REGION Network 41: FIT-503 LOW
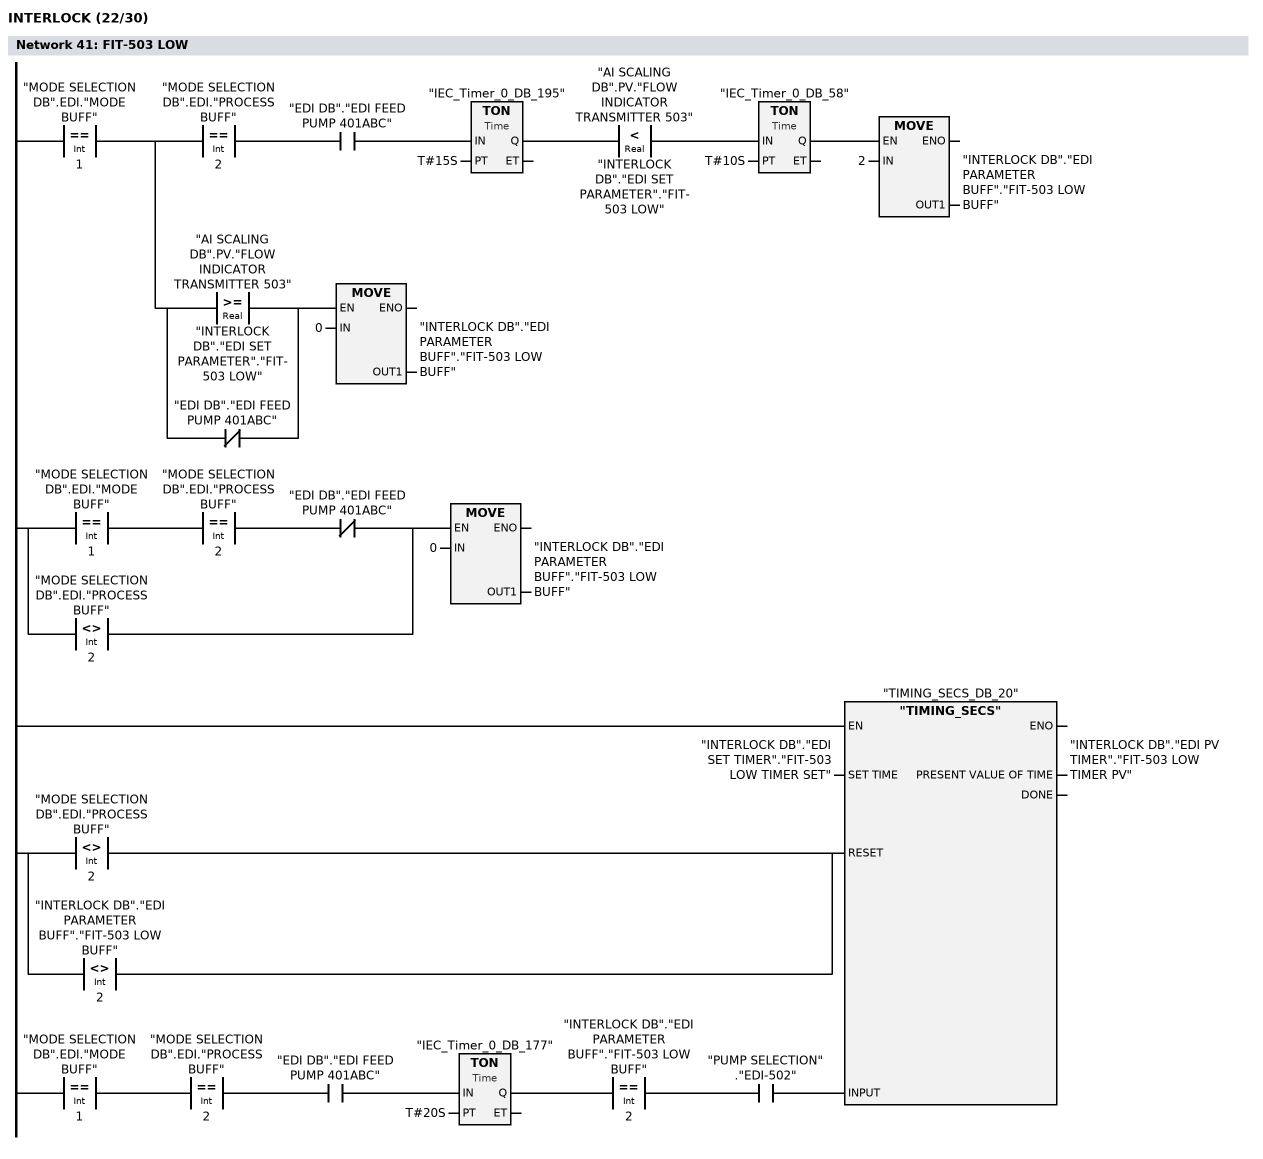
   RUNG wire#powerrail
      { S7_Templates := "SrcType := Int" } EQ_Contact(in1 := "MODE SELECTION DB".EDI."MODE BUFF", in2 := 1)
      wire#w1
      { S7_Templates := "SrcType := Int" } EQ_Contact(in1 := "MODE SELECTION DB".EDI."PROCESS BUFF", in2 := 2)
      Contact( "EDI DB"."EDI FEED PUMP 401ABC" )
      { S7_Templates := "time_type := Time" } "IEC_Timer_0_DB_195".TON(pt := T#15S, et =>)
      { S7_Templates := "SrcType := Real" } LT_Contact(in1 := "AI SCALING DB".PV."FLOW INDICATOR TRANSMITTER 503", in2 := "INTERLOCK DB"."EDI SET PARAMETER"."FIT-503 LOW")
      { S7_Templates := "time_type := Time" } "IEC_Timer_0_DB_58".TON(pt := T#10S, et =>)
      Move(in := 2, out1 => "INTERLOCK DB"."EDI PARAMETER BUFF"."FIT-503 LOW BUFF")
   END_RUNG
   RUNG wire#w1
      { S7_Templates := "SrcType := Real" } GE_Contact(in1 := "AI SCALING DB".PV."FLOW INDICATOR TRANSMITTER 503", in2 := "INTERLOCK DB"."EDI SET PARAMETER"."FIT-503 LOW")
      wire#w2
      Move(in := 0, out1 => "INTERLOCK DB"."EDI PARAMETER BUFF"."FIT-503 LOW BUFF")
   END_RUNG
   RUNG wire#w1
      I_Contact( "EDI DB"."EDI FEED PUMP 401ABC" )
   END_RUNG wire#w2
   RUNG wire#powerrail
      { S7_Templates := "SrcType := Int" } EQ_Contact(in1 := "MODE SELECTION DB".EDI."MODE BUFF", in2 := 1)
      { S7_Templates := "SrcType := Int" } EQ_Contact(in1 := "MODE SELECTION DB".EDI."PROCESS BUFF", in2 := 2)
      I_Contact( "EDI DB"."EDI FEED PUMP 401ABC" )
      wire#w3
      Move(in := 0, out1 => "INTERLOCK DB"."EDI PARAMETER BUFF"."FIT-503 LOW BUFF")
   END_RUNG
   RUNG wire#powerrail
      { S7_Templates := "SrcType := Int" } NE_Contact(in1 := "MODE SELECTION DB".EDI."PROCESS BUFF", in2 := 2)
   END_RUNG wire#w3
   RUNG wire#powerrail
      "TIMING_SECS_DB_20"(RESET := wire#w4, INPUT := wire#w5, "SET TIME" := "INTERLOCK DB"."EDI SET TIMER"."FIT-503 LOW TIMER SET", "PRESENT VALUE OF TIME" => "INTERLOCK DB"."EDI PV TIMER"."FIT-503 LOW TIMER PV", DONE =>)
   END_RUNG
   RUNG wire#powerrail
      { S7_Templates := "SrcType := Int" } NE_Contact(in1 := "MODE SELECTION DB".EDI."PROCESS BUFF", in2 := 2)
   END_RUNG wire#w4
   RUNG wire#powerrail
      { S7_Templates := "SrcType := Int" } NE_Contact(in1 := "INTERLOCK DB"."EDI PARAMETER BUFF"."FIT-503 LOW BUFF", in2 := 2)
   END_RUNG wire#w4
   RUNG wire#powerrail
      { S7_Templates := "SrcType := Int" } EQ_Contact(in1 := "MODE SELECTION DB".EDI."MODE BUFF", in2 := 1)
      { S7_Templates := "SrcType := Int" } EQ_Contact(in1 := "MODE SELECTION DB".EDI."PROCESS BUFF", in2 := 2)
      Contact( "EDI DB"."EDI FEED PUMP 401ABC" )
      { S7_Templates := "time_type := Time" } "IEC_Timer_0_DB_177".TON(pt := T#20S, et =>)
      { S7_Templates := "SrcType := Int" } EQ_Contact(in1 := "INTERLOCK DB"."EDI PARAMETER BUFF"."FIT-503 LOW BUFF", in2 := 2)
      Contact( "PUMP SELECTION"."EDI-502" )
   END_RUNG wire#w5
   // the same network as SCL:
   #_w1 := "MODE SELECTION DB".EDI."MODE BUFF" = 1;
   "IEC_Timer_0_DB_195".TON(IN := #_w1 AND ("MODE SELECTION DB".EDI."PROCESS BUFF" = 2) AND "EDI DB"."EDI FEED PUMP 401ABC",
                           PT := T#15S);
   "IEC_Timer_0_DB_58".TON(IN := "IEC_Timer_0_DB_195".Q AND ("AI SCALING DB".PV."FLOW INDICATOR TRANSMITTER 503" < "INTERLOCK DB"."EDI SET PARAMETER"."FIT-503 LOW"),
                           PT := T#10S);
   IF "IEC_Timer_0_DB_58".Q THEN "INTERLOCK DB"."EDI PARAMETER BUFF"."FIT-503 LOW BUFF" := 2; END_IF;
   IF #_w1 AND (("AI SCALING DB".PV."FLOW INDICATOR TRANSMITTER 503" >= "INTERLOCK DB"."EDI SET PARAMETER"."FIT-503 LOW") OR NOT "EDI DB"."EDI FEED PUMP 401ABC") THEN
       "INTERLOCK DB"."EDI PARAMETER BUFF"."FIT-503 LOW BUFF" := 0;
   END_IF;
   IF (("MODE SELECTION DB".EDI."MODE BUFF" = 1) AND ("MODE SELECTION DB".EDI."PROCESS BUFF" = 2) AND NOT "EDI DB"."EDI FEED PUMP 401ABC") OR ("MODE SELECTION DB".EDI."PROCESS BUFF" <> 2) THEN
       "INTERLOCK DB"."EDI PARAMETER BUFF"."FIT-503 LOW BUFF" := 0;
   END_IF;
   "IEC_Timer_0_DB_177".TON(IN := ("MODE SELECTION DB".EDI."MODE BUFF" = 1) AND ("MODE SELECTION DB".EDI."PROCESS BUFF" = 2) AND "EDI DB"."EDI FEED PUMP 401ABC",
                           PT := T#20S);
   "TIMING_SECS_DB_20"("SET TIME" := "INTERLOCK DB"."EDI SET TIMER"."FIT-503 LOW TIMER SET",   // "TIMING_SECS"
                       RESET := ("MODE SELECTION DB".EDI."PROCESS BUFF" <> 2) OR ("INTERLOCK DB"."EDI PARAMETER BUFF"."FIT-503 LOW BUFF" <> 2),
                       INPUT := "IEC_Timer_0_DB_177".Q AND ("INTERLOCK DB"."EDI PARAMETER BUFF"."FIT-503 LOW BUFF" = 2) AND "PUMP SELECTION"."EDI-502",
                       "PRESENT VALUE OF TIME" => "INTERLOCK DB"."EDI PV TIMER"."FIT-503 LOW TIMER PV");
END_REGION

REGION Network 42: FIT-504 LOW
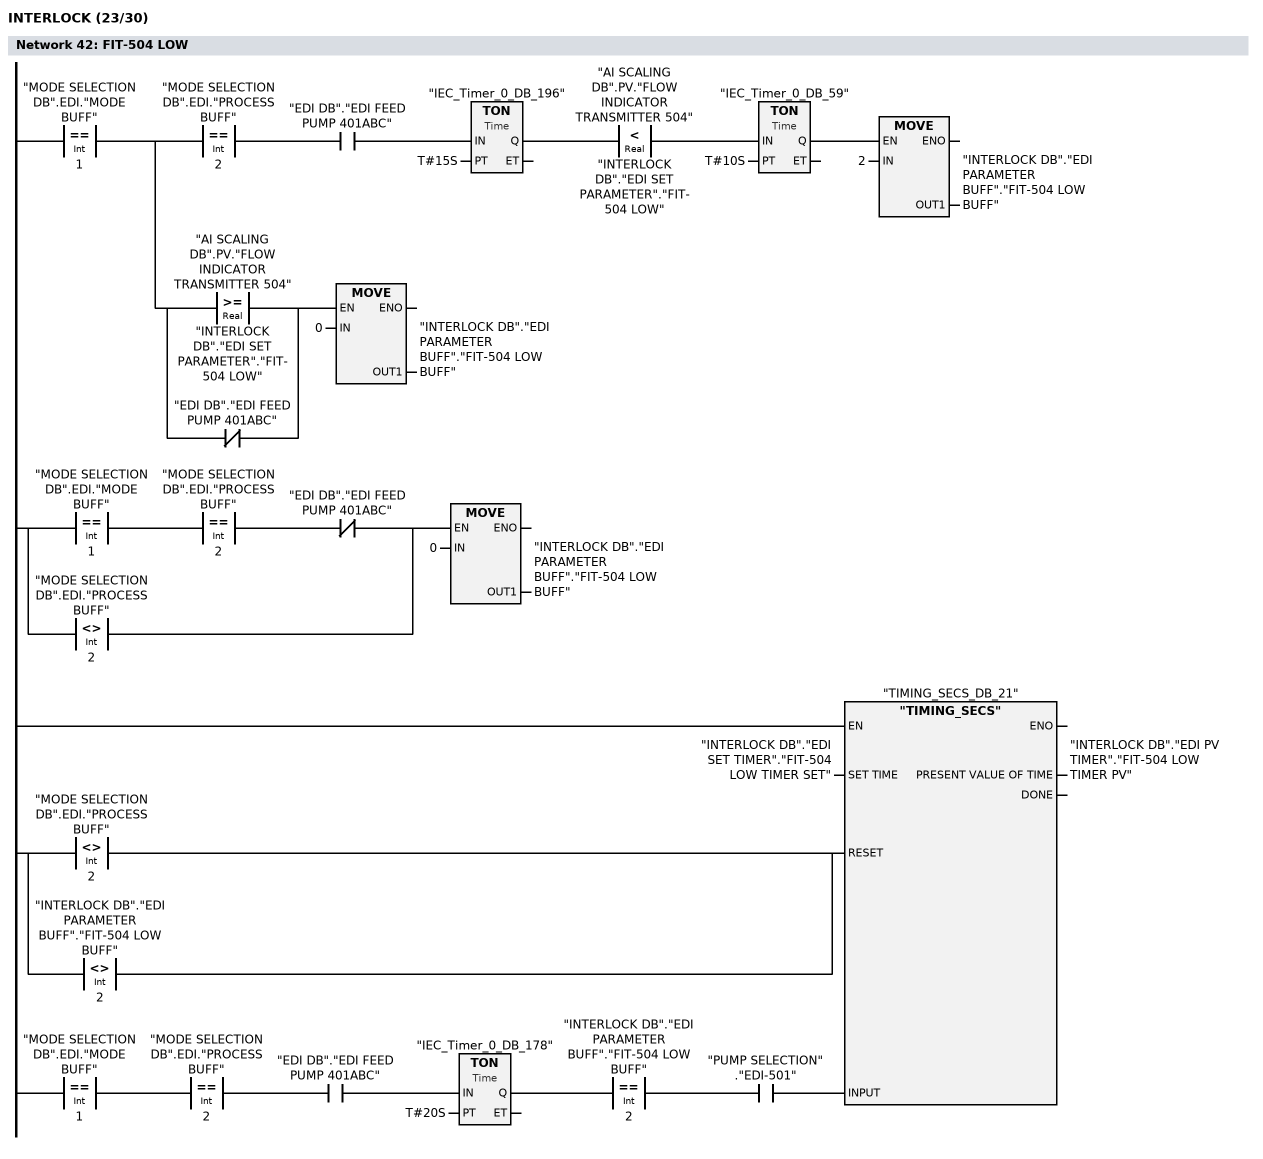
   RUNG wire#powerrail
      { S7_Templates := "SrcType := Int" } EQ_Contact(in1 := "MODE SELECTION DB".EDI."MODE BUFF", in2 := 1)
      wire#w1
      { S7_Templates := "SrcType := Int" } EQ_Contact(in1 := "MODE SELECTION DB".EDI."PROCESS BUFF", in2 := 2)
      Contact( "EDI DB"."EDI FEED PUMP 401ABC" )
      { S7_Templates := "time_type := Time" } "IEC_Timer_0_DB_196".TON(pt := T#15S, et =>)
      { S7_Templates := "SrcType := Real" } LT_Contact(in1 := "AI SCALING DB".PV."FLOW INDICATOR TRANSMITTER 504", in2 := "INTERLOCK DB"."EDI SET PARAMETER"."FIT-504 LOW")
      { S7_Templates := "time_type := Time" } "IEC_Timer_0_DB_59".TON(pt := T#10S, et =>)
      Move(in := 2, out1 => "INTERLOCK DB"."EDI PARAMETER BUFF"."FIT-504 LOW BUFF")
   END_RUNG
   RUNG wire#w1
      { S7_Templates := "SrcType := Real" } GE_Contact(in1 := "AI SCALING DB".PV."FLOW INDICATOR TRANSMITTER 504", in2 := "INTERLOCK DB"."EDI SET PARAMETER"."FIT-504 LOW")
      wire#w2
      Move(in := 0, out1 => "INTERLOCK DB"."EDI PARAMETER BUFF"."FIT-504 LOW BUFF")
   END_RUNG
   RUNG wire#w1
      I_Contact( "EDI DB"."EDI FEED PUMP 401ABC" )
   END_RUNG wire#w2
   RUNG wire#powerrail
      { S7_Templates := "SrcType := Int" } EQ_Contact(in1 := "MODE SELECTION DB".EDI."MODE BUFF", in2 := 1)
      { S7_Templates := "SrcType := Int" } EQ_Contact(in1 := "MODE SELECTION DB".EDI."PROCESS BUFF", in2 := 2)
      I_Contact( "EDI DB"."EDI FEED PUMP 401ABC" )
      wire#w3
      Move(in := 0, out1 => "INTERLOCK DB"."EDI PARAMETER BUFF"."FIT-504 LOW BUFF")
   END_RUNG
   RUNG wire#powerrail
      { S7_Templates := "SrcType := Int" } NE_Contact(in1 := "MODE SELECTION DB".EDI."PROCESS BUFF", in2 := 2)
   END_RUNG wire#w3
   RUNG wire#powerrail
      "TIMING_SECS_DB_21"(RESET := wire#w4, INPUT := wire#w5, "SET TIME" := "INTERLOCK DB"."EDI SET TIMER"."FIT-504 LOW TIMER SET", "PRESENT VALUE OF TIME" => "INTERLOCK DB"."EDI PV TIMER"."FIT-504 LOW TIMER PV", DONE =>)
   END_RUNG
   RUNG wire#powerrail
      { S7_Templates := "SrcType := Int" } NE_Contact(in1 := "MODE SELECTION DB".EDI."PROCESS BUFF", in2 := 2)
   END_RUNG wire#w4
   RUNG wire#powerrail
      { S7_Templates := "SrcType := Int" } NE_Contact(in1 := "INTERLOCK DB"."EDI PARAMETER BUFF"."FIT-504 LOW BUFF", in2 := 2)
   END_RUNG wire#w4
   RUNG wire#powerrail
      { S7_Templates := "SrcType := Int" } EQ_Contact(in1 := "MODE SELECTION DB".EDI."MODE BUFF", in2 := 1)
      { S7_Templates := "SrcType := Int" } EQ_Contact(in1 := "MODE SELECTION DB".EDI."PROCESS BUFF", in2 := 2)
      Contact( "EDI DB"."EDI FEED PUMP 401ABC" )
      { S7_Templates := "time_type := Time" } "IEC_Timer_0_DB_178".TON(pt := T#20S, et =>)
      { S7_Templates := "SrcType := Int" } EQ_Contact(in1 := "INTERLOCK DB"."EDI PARAMETER BUFF"."FIT-504 LOW BUFF", in2 := 2)
      Contact( "PUMP SELECTION"."EDI-501" )
   END_RUNG wire#w5
   // the same network as SCL:
   #_w1 := "MODE SELECTION DB".EDI."MODE BUFF" = 1;
   "IEC_Timer_0_DB_196".TON(IN := #_w1 AND ("MODE SELECTION DB".EDI."PROCESS BUFF" = 2) AND "EDI DB"."EDI FEED PUMP 401ABC",
                           PT := T#15S);
   "IEC_Timer_0_DB_59".TON(IN := "IEC_Timer_0_DB_196".Q AND ("AI SCALING DB".PV."FLOW INDICATOR TRANSMITTER 504" < "INTERLOCK DB"."EDI SET PARAMETER"."FIT-504 LOW"),
                           PT := T#10S);
   IF "IEC_Timer_0_DB_59".Q THEN "INTERLOCK DB"."EDI PARAMETER BUFF"."FIT-504 LOW BUFF" := 2; END_IF;
   IF #_w1 AND (("AI SCALING DB".PV."FLOW INDICATOR TRANSMITTER 504" >= "INTERLOCK DB"."EDI SET PARAMETER"."FIT-504 LOW") OR NOT "EDI DB"."EDI FEED PUMP 401ABC") THEN
       "INTERLOCK DB"."EDI PARAMETER BUFF"."FIT-504 LOW BUFF" := 0;
   END_IF;
   IF (("MODE SELECTION DB".EDI."MODE BUFF" = 1) AND ("MODE SELECTION DB".EDI."PROCESS BUFF" = 2) AND NOT "EDI DB"."EDI FEED PUMP 401ABC") OR ("MODE SELECTION DB".EDI."PROCESS BUFF" <> 2) THEN
       "INTERLOCK DB"."EDI PARAMETER BUFF"."FIT-504 LOW BUFF" := 0;
   END_IF;
   "IEC_Timer_0_DB_178".TON(IN := ("MODE SELECTION DB".EDI."MODE BUFF" = 1) AND ("MODE SELECTION DB".EDI."PROCESS BUFF" = 2) AND "EDI DB"."EDI FEED PUMP 401ABC",
                           PT := T#20S);
   "TIMING_SECS_DB_21"("SET TIME" := "INTERLOCK DB"."EDI SET TIMER"."FIT-504 LOW TIMER SET",   // "TIMING_SECS"
                       RESET := ("MODE SELECTION DB".EDI."PROCESS BUFF" <> 2) OR ("INTERLOCK DB"."EDI PARAMETER BUFF"."FIT-504 LOW BUFF" <> 2),
                       INPUT := "IEC_Timer_0_DB_178".Q AND ("INTERLOCK DB"."EDI PARAMETER BUFF"."FIT-504 LOW BUFF" = 2) AND "PUMP SELECTION"."EDI-501",
                       "PRESENT VALUE OF TIME" => "INTERLOCK DB"."EDI PV TIMER"."FIT-504 LOW TIMER PV");
END_REGION

REGION Network 43: FIT-505 LOW / HIGH
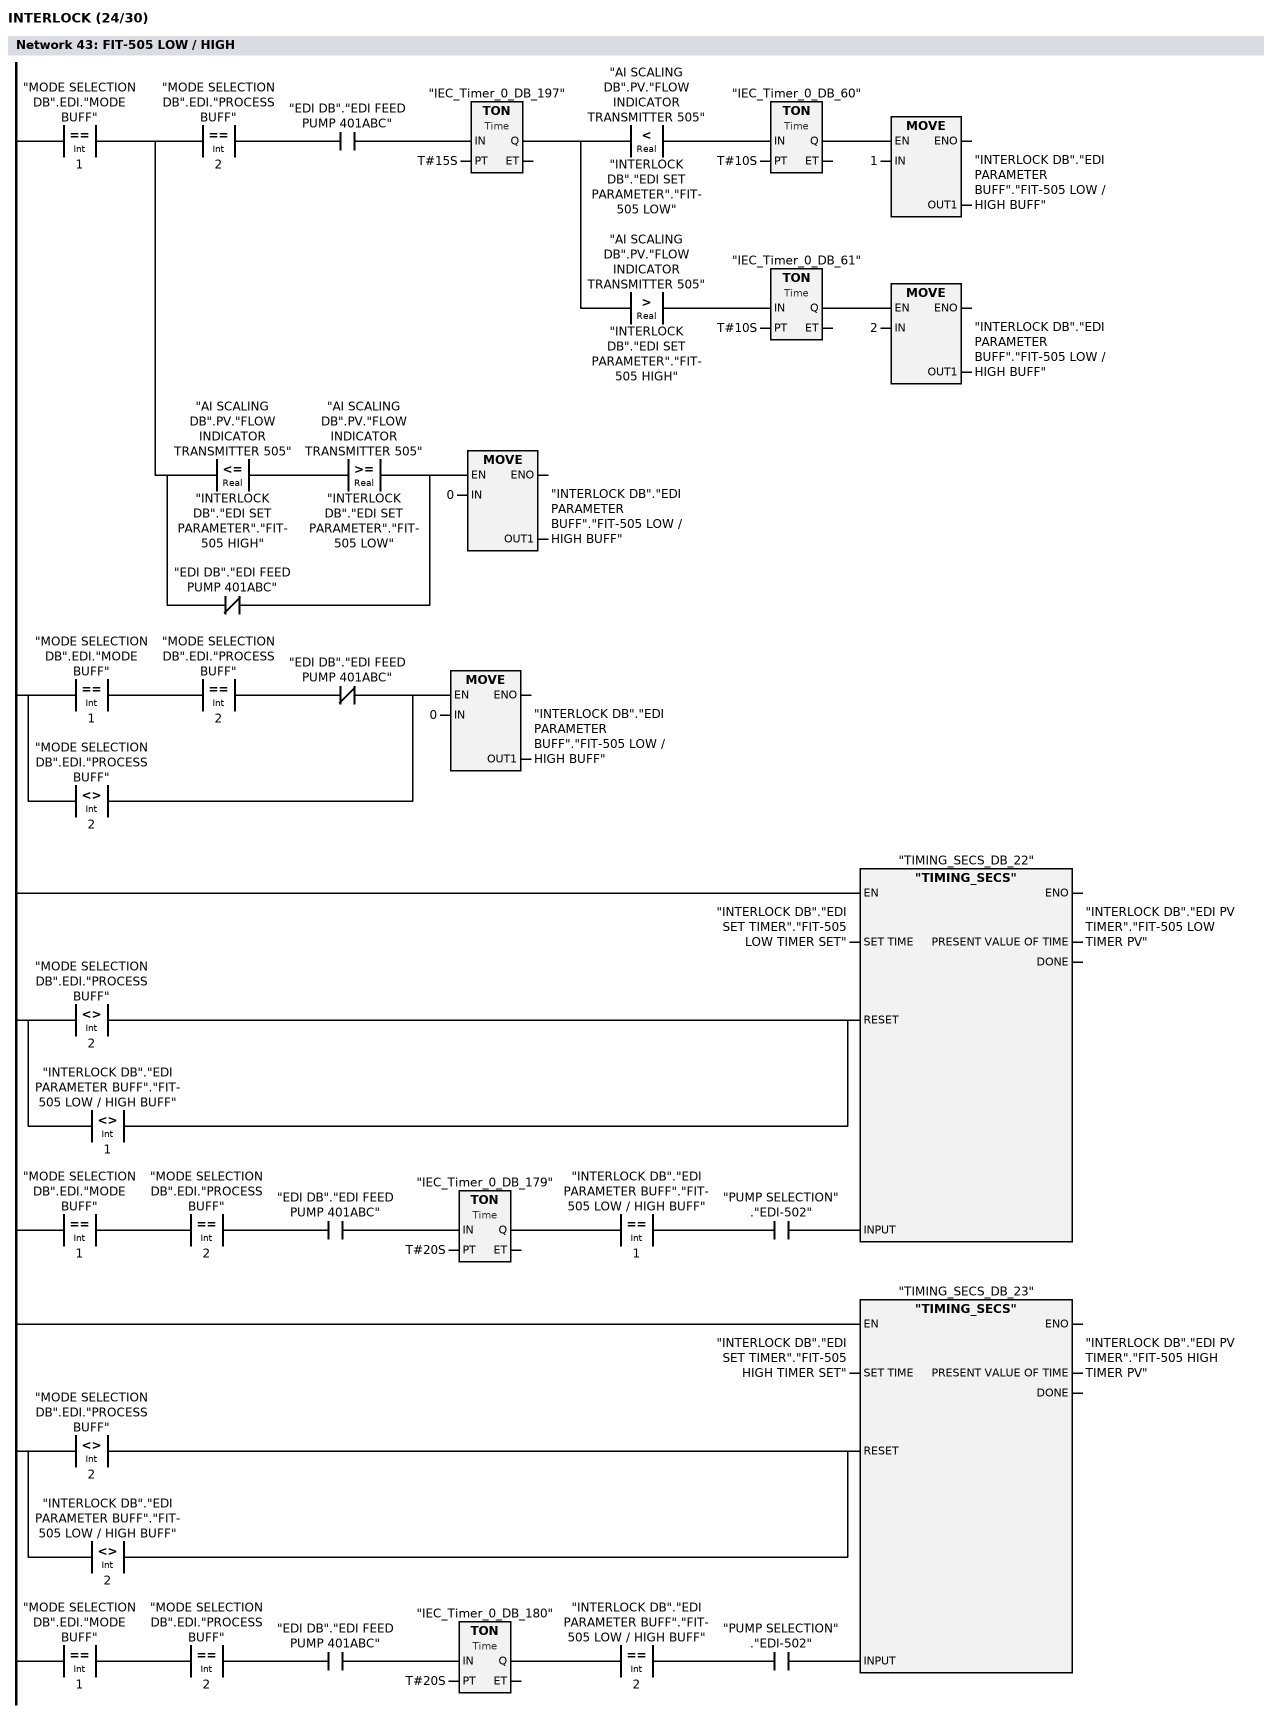
   RUNG wire#powerrail
      { S7_Templates := "SrcType := Int" } EQ_Contact(in1 := "MODE SELECTION DB".EDI."MODE BUFF", in2 := 1)
      wire#w1
      { S7_Templates := "SrcType := Int" } EQ_Contact(in1 := "MODE SELECTION DB".EDI."PROCESS BUFF", in2 := 2)
      Contact( "EDI DB"."EDI FEED PUMP 401ABC" )
      { S7_Templates := "time_type := Time" } "IEC_Timer_0_DB_197".TON(pt := T#15S, et =>)
      wire#w2
      { S7_Templates := "SrcType := Real" } LT_Contact(in1 := "AI SCALING DB".PV."FLOW INDICATOR TRANSMITTER 505", in2 := "INTERLOCK DB"."EDI SET PARAMETER"."FIT-505 LOW")
      { S7_Templates := "time_type := Time" } "IEC_Timer_0_DB_60".TON(pt := T#10S, et =>)
      Move(in := 1, out1 => "INTERLOCK DB"."EDI PARAMETER BUFF"."FIT-505 LOW / HIGH BUFF")
   END_RUNG
   RUNG wire#w2
      { S7_Templates := "SrcType := Real" } GT_Contact(in1 := "AI SCALING DB".PV."FLOW INDICATOR TRANSMITTER 505", in2 := "INTERLOCK DB"."EDI SET PARAMETER"."FIT-505 HIGH")
      { S7_Templates := "time_type := Time" } "IEC_Timer_0_DB_61".TON(pt := T#10S, et =>)
      Move(in := 2, out1 => "INTERLOCK DB"."EDI PARAMETER BUFF"."FIT-505 LOW / HIGH BUFF")
   END_RUNG
   RUNG wire#w1
      { S7_Templates := "SrcType := Real" } LE_Contact(in1 := "AI SCALING DB".PV."FLOW INDICATOR TRANSMITTER 505", in2 := "INTERLOCK DB"."EDI SET PARAMETER"."FIT-505 HIGH")
      { S7_Templates := "SrcType := Real" } GE_Contact(in1 := "AI SCALING DB".PV."FLOW INDICATOR TRANSMITTER 505", in2 := "INTERLOCK DB"."EDI SET PARAMETER"."FIT-505 LOW")
      wire#w3
      Move(in := 0, out1 => "INTERLOCK DB"."EDI PARAMETER BUFF"."FIT-505 LOW / HIGH BUFF")
   END_RUNG
   RUNG wire#w1
      I_Contact( "EDI DB"."EDI FEED PUMP 401ABC" )
   END_RUNG wire#w3
   RUNG wire#powerrail
      { S7_Templates := "SrcType := Int" } EQ_Contact(in1 := "MODE SELECTION DB".EDI."MODE BUFF", in2 := 1)
      { S7_Templates := "SrcType := Int" } EQ_Contact(in1 := "MODE SELECTION DB".EDI."PROCESS BUFF", in2 := 2)
      I_Contact( "EDI DB"."EDI FEED PUMP 401ABC" )
      wire#w4
      Move(in := 0, out1 => "INTERLOCK DB"."EDI PARAMETER BUFF"."FIT-505 LOW / HIGH BUFF")
   END_RUNG
   RUNG wire#powerrail
      { S7_Templates := "SrcType := Int" } NE_Contact(in1 := "MODE SELECTION DB".EDI."PROCESS BUFF", in2 := 2)
   END_RUNG wire#w4
   RUNG wire#powerrail
      "TIMING_SECS_DB_22"(RESET := wire#w5, INPUT := wire#w6, "SET TIME" := "INTERLOCK DB"."EDI SET TIMER"."FIT-505 LOW TIMER SET", "PRESENT VALUE OF TIME" => "INTERLOCK DB"."EDI PV TIMER"."FIT-505 LOW TIMER PV", DONE =>)
   END_RUNG
   RUNG wire#powerrail
      { S7_Templates := "SrcType := Int" } NE_Contact(in1 := "MODE SELECTION DB".EDI."PROCESS BUFF", in2 := 2)
   END_RUNG wire#w5
   RUNG wire#powerrail
      { S7_Templates := "SrcType := Int" } NE_Contact(in1 := "INTERLOCK DB"."EDI PARAMETER BUFF"."FIT-505 LOW / HIGH BUFF", in2 := 1)
   END_RUNG wire#w5
   RUNG wire#powerrail
      { S7_Templates := "SrcType := Int" } EQ_Contact(in1 := "MODE SELECTION DB".EDI."MODE BUFF", in2 := 1)
      { S7_Templates := "SrcType := Int" } EQ_Contact(in1 := "MODE SELECTION DB".EDI."PROCESS BUFF", in2 := 2)
      Contact( "EDI DB"."EDI FEED PUMP 401ABC" )
      { S7_Templates := "time_type := Time" } "IEC_Timer_0_DB_179".TON(pt := T#20S, et =>)
      { S7_Templates := "SrcType := Int" } EQ_Contact(in1 := "INTERLOCK DB"."EDI PARAMETER BUFF"."FIT-505 LOW / HIGH BUFF", in2 := 1)
      Contact( "PUMP SELECTION"."EDI-502" )
   END_RUNG wire#w6
   RUNG wire#powerrail
      "TIMING_SECS_DB_23"(RESET := wire#w7, INPUT := wire#w8, "SET TIME" := "INTERLOCK DB"."EDI SET TIMER"."FIT-505 HIGH TIMER SET", "PRESENT VALUE OF TIME" => "INTERLOCK DB"."EDI PV TIMER"."FIT-505 HIGH TIMER PV", DONE =>)
   END_RUNG
   RUNG wire#powerrail
      { S7_Templates := "SrcType := Int" } NE_Contact(in1 := "MODE SELECTION DB".EDI."PROCESS BUFF", in2 := 2)
   END_RUNG wire#w7
   RUNG wire#powerrail
      { S7_Templates := "SrcType := Int" } NE_Contact(in1 := "INTERLOCK DB"."EDI PARAMETER BUFF"."FIT-505 LOW / HIGH BUFF", in2 := 2)
   END_RUNG wire#w7
   RUNG wire#powerrail
      { S7_Templates := "SrcType := Int" } EQ_Contact(in1 := "MODE SELECTION DB".EDI."MODE BUFF", in2 := 1)
      { S7_Templates := "SrcType := Int" } EQ_Contact(in1 := "MODE SELECTION DB".EDI."PROCESS BUFF", in2 := 2)
      Contact( "EDI DB"."EDI FEED PUMP 401ABC" )
      { S7_Templates := "time_type := Time" } "IEC_Timer_0_DB_180".TON(pt := T#20S, et =>)
      { S7_Templates := "SrcType := Int" } EQ_Contact(in1 := "INTERLOCK DB"."EDI PARAMETER BUFF"."FIT-505 LOW / HIGH BUFF", in2 := 2)
      Contact( "PUMP SELECTION"."EDI-502" )
   END_RUNG wire#w8
   // the same network as SCL:
   #_w1 := "MODE SELECTION DB".EDI."MODE BUFF" = 1;
   "IEC_Timer_0_DB_197".TON(IN := #_w1 AND ("MODE SELECTION DB".EDI."PROCESS BUFF" = 2) AND "EDI DB"."EDI FEED PUMP 401ABC",
                           PT := T#15S);
   "IEC_Timer_0_DB_60".TON(IN := "IEC_Timer_0_DB_197".Q AND ("AI SCALING DB".PV."FLOW INDICATOR TRANSMITTER 505" < "INTERLOCK DB"."EDI SET PARAMETER"."FIT-505 LOW"),
                           PT := T#10S);
   IF "IEC_Timer_0_DB_60".Q THEN "INTERLOCK DB"."EDI PARAMETER BUFF"."FIT-505 LOW / HIGH BUFF" := 1; END_IF;
   "IEC_Timer_0_DB_61".TON(IN := "IEC_Timer_0_DB_197".Q AND ("AI SCALING DB".PV."FLOW INDICATOR TRANSMITTER 505" > "INTERLOCK DB"."EDI SET PARAMETER"."FIT-505 HIGH"),
                           PT := T#10S);
   IF "IEC_Timer_0_DB_61".Q THEN "INTERLOCK DB"."EDI PARAMETER BUFF"."FIT-505 LOW / HIGH BUFF" := 2; END_IF;
   IF #_w1 AND ((("AI SCALING DB".PV."FLOW INDICATOR TRANSMITTER 505" <= "INTERLOCK DB"."EDI SET PARAMETER"."FIT-505 HIGH") AND ("AI SCALING DB".PV."FLOW INDICATOR TRANSMITTER 505" >= "INTERLOCK DB"."EDI SET PARAMETER"."FIT-505 LOW")) OR NOT "EDI DB"."EDI FEED PUMP 401ABC") THEN
       "INTERLOCK DB"."EDI PARAMETER BUFF"."FIT-505 LOW / HIGH BUFF" := 0;
   END_IF;
   IF (("MODE SELECTION DB".EDI."MODE BUFF" = 1) AND ("MODE SELECTION DB".EDI."PROCESS BUFF" = 2) AND NOT "EDI DB"."EDI FEED PUMP 401ABC") OR ("MODE SELECTION DB".EDI."PROCESS BUFF" <> 2) THEN
       "INTERLOCK DB"."EDI PARAMETER BUFF"."FIT-505 LOW / HIGH BUFF" := 0;
   END_IF;
   "IEC_Timer_0_DB_179".TON(IN := ("MODE SELECTION DB".EDI."MODE BUFF" = 1) AND ("MODE SELECTION DB".EDI."PROCESS BUFF" = 2) AND "EDI DB"."EDI FEED PUMP 401ABC",
                           PT := T#20S);
   "TIMING_SECS_DB_22"("SET TIME" := "INTERLOCK DB"."EDI SET TIMER"."FIT-505 LOW TIMER SET",   // "TIMING_SECS"
                       RESET := ("MODE SELECTION DB".EDI."PROCESS BUFF" <> 2) OR ("INTERLOCK DB"."EDI PARAMETER BUFF"."FIT-505 LOW / HIGH BUFF" <> 1),
                       INPUT := "IEC_Timer_0_DB_179".Q AND ("INTERLOCK DB"."EDI PARAMETER BUFF"."FIT-505 LOW / HIGH BUFF" = 1) AND "PUMP SELECTION"."EDI-502",
                       "PRESENT VALUE OF TIME" => "INTERLOCK DB"."EDI PV TIMER"."FIT-505 LOW TIMER PV");
   "IEC_Timer_0_DB_180".TON(IN := ("MODE SELECTION DB".EDI."MODE BUFF" = 1) AND ("MODE SELECTION DB".EDI."PROCESS BUFF" = 2) AND "EDI DB"."EDI FEED PUMP 401ABC",
                           PT := T#20S);
   "TIMING_SECS_DB_23"("SET TIME" := "INTERLOCK DB"."EDI SET TIMER"."FIT-505 HIGH TIMER SET",   // "TIMING_SECS"
                       RESET := ("MODE SELECTION DB".EDI."PROCESS BUFF" <> 2) OR ("INTERLOCK DB"."EDI PARAMETER BUFF"."FIT-505 LOW / HIGH BUFF" <> 2),
                       INPUT := "IEC_Timer_0_DB_180".Q AND ("INTERLOCK DB"."EDI PARAMETER BUFF"."FIT-505 LOW / HIGH BUFF" = 2) AND "PUMP SELECTION"."EDI-502",
                       "PRESENT VALUE OF TIME" => "INTERLOCK DB"."EDI PV TIMER"."FIT-505 HIGH TIMER PV");
END_REGION

REGION Network 44: FIT-506 LOW / HIGH
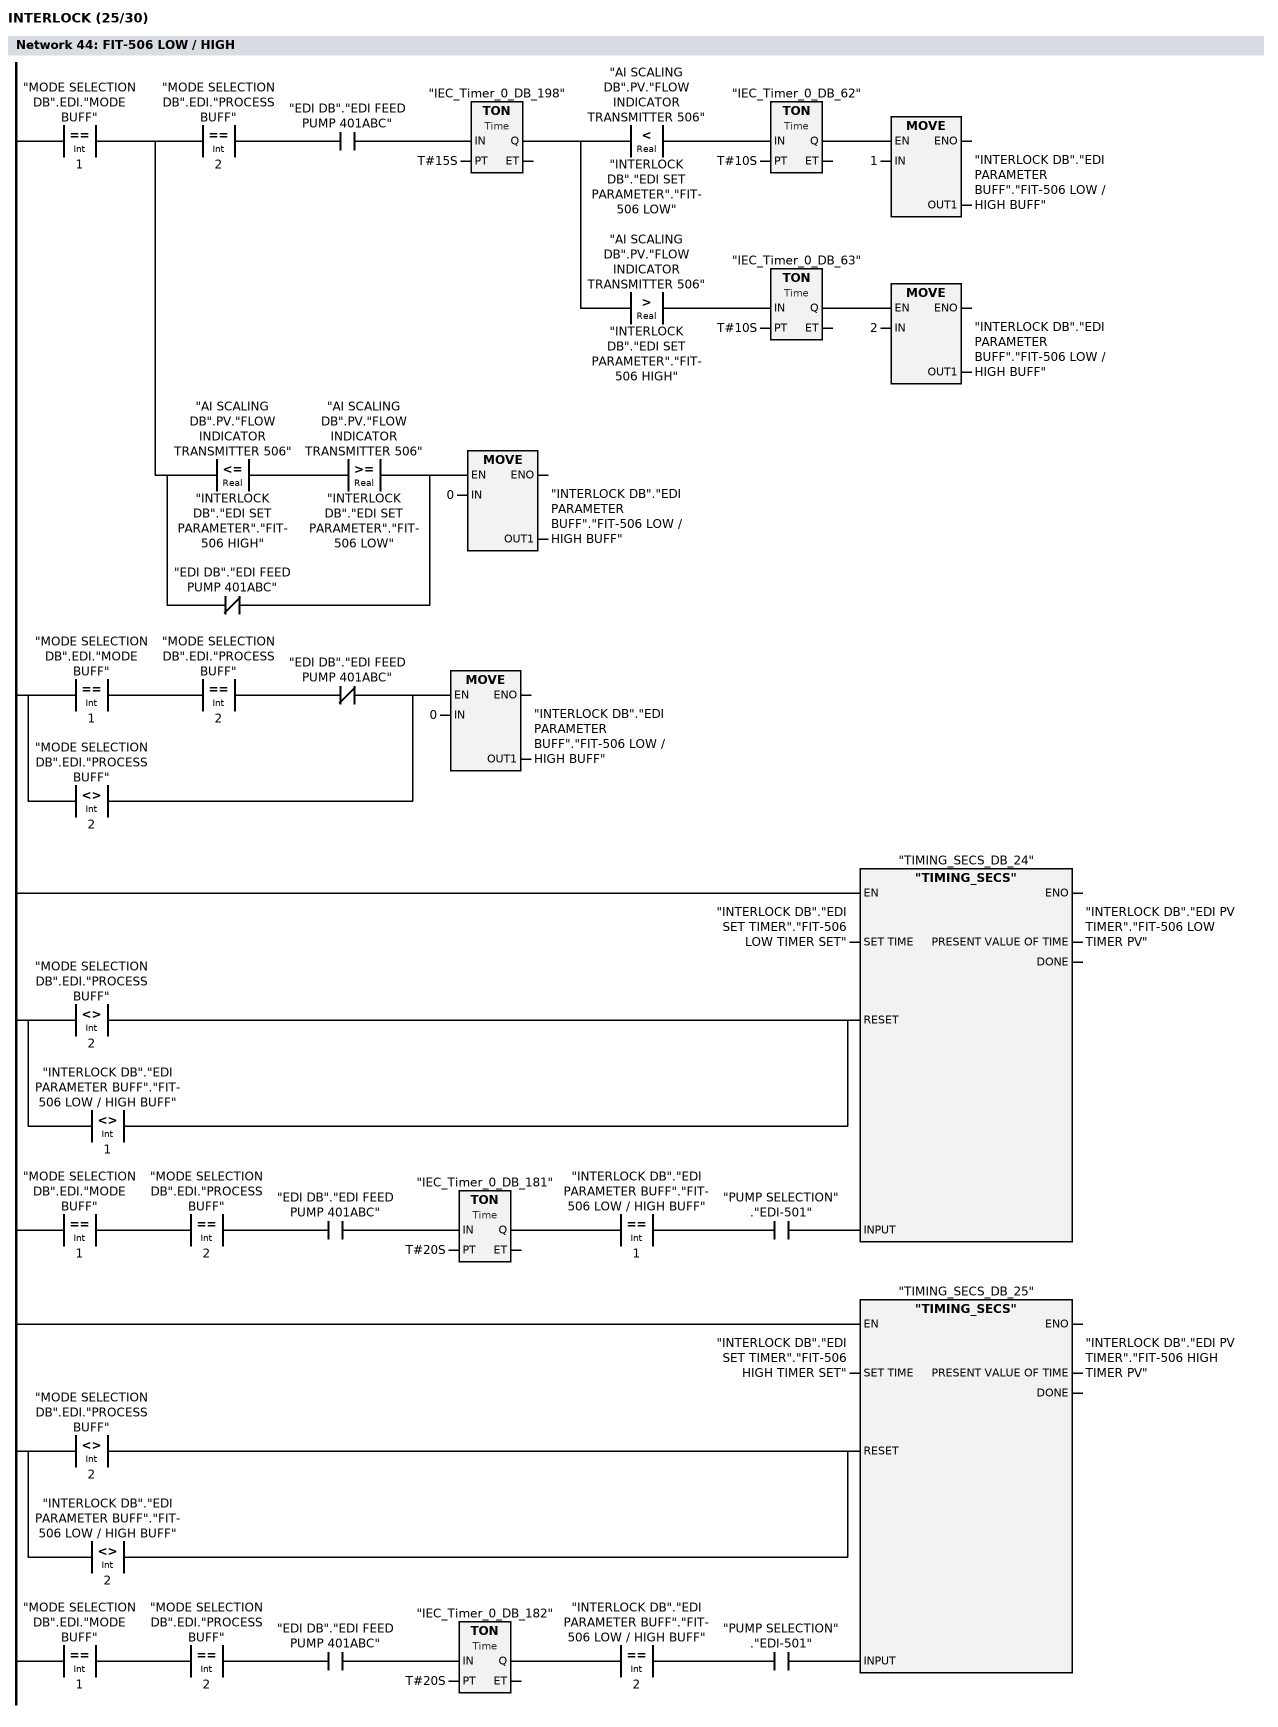
   RUNG wire#powerrail
      { S7_Templates := "SrcType := Int" } EQ_Contact(in1 := "MODE SELECTION DB".EDI."MODE BUFF", in2 := 1)
      wire#w1
      { S7_Templates := "SrcType := Int" } EQ_Contact(in1 := "MODE SELECTION DB".EDI."PROCESS BUFF", in2 := 2)
      Contact( "EDI DB"."EDI FEED PUMP 401ABC" )
      { S7_Templates := "time_type := Time" } "IEC_Timer_0_DB_198".TON(pt := T#15S, et =>)
      wire#w2
      { S7_Templates := "SrcType := Real" } LT_Contact(in1 := "AI SCALING DB".PV."FLOW INDICATOR TRANSMITTER 506", in2 := "INTERLOCK DB"."EDI SET PARAMETER"."FIT-506 LOW")
      { S7_Templates := "time_type := Time" } "IEC_Timer_0_DB_62".TON(pt := T#10S, et =>)
      Move(in := 1, out1 => "INTERLOCK DB"."EDI PARAMETER BUFF"."FIT-506 LOW / HIGH BUFF")
   END_RUNG
   RUNG wire#w2
      { S7_Templates := "SrcType := Real" } GT_Contact(in1 := "AI SCALING DB".PV."FLOW INDICATOR TRANSMITTER 506", in2 := "INTERLOCK DB"."EDI SET PARAMETER"."FIT-506 HIGH")
      { S7_Templates := "time_type := Time" } "IEC_Timer_0_DB_63".TON(pt := T#10S, et =>)
      Move(in := 2, out1 => "INTERLOCK DB"."EDI PARAMETER BUFF"."FIT-506 LOW / HIGH BUFF")
   END_RUNG
   RUNG wire#w1
      { S7_Templates := "SrcType := Real" } LE_Contact(in1 := "AI SCALING DB".PV."FLOW INDICATOR TRANSMITTER 506", in2 := "INTERLOCK DB"."EDI SET PARAMETER"."FIT-506 HIGH")
      { S7_Templates := "SrcType := Real" } GE_Contact(in1 := "AI SCALING DB".PV."FLOW INDICATOR TRANSMITTER 506", in2 := "INTERLOCK DB"."EDI SET PARAMETER"."FIT-506 LOW")
      wire#w3
      Move(in := 0, out1 => "INTERLOCK DB"."EDI PARAMETER BUFF"."FIT-506 LOW / HIGH BUFF")
   END_RUNG
   RUNG wire#w1
      I_Contact( "EDI DB"."EDI FEED PUMP 401ABC" )
   END_RUNG wire#w3
   RUNG wire#powerrail
      { S7_Templates := "SrcType := Int" } EQ_Contact(in1 := "MODE SELECTION DB".EDI."MODE BUFF", in2 := 1)
      { S7_Templates := "SrcType := Int" } EQ_Contact(in1 := "MODE SELECTION DB".EDI."PROCESS BUFF", in2 := 2)
      I_Contact( "EDI DB"."EDI FEED PUMP 401ABC" )
      wire#w4
      Move(in := 0, out1 => "INTERLOCK DB"."EDI PARAMETER BUFF"."FIT-506 LOW / HIGH BUFF")
   END_RUNG
   RUNG wire#powerrail
      { S7_Templates := "SrcType := Int" } NE_Contact(in1 := "MODE SELECTION DB".EDI."PROCESS BUFF", in2 := 2)
   END_RUNG wire#w4
   RUNG wire#powerrail
      "TIMING_SECS_DB_24"(RESET := wire#w5, INPUT := wire#w6, "SET TIME" := "INTERLOCK DB"."EDI SET TIMER"."FIT-506 LOW TIMER SET", "PRESENT VALUE OF TIME" => "INTERLOCK DB"."EDI PV TIMER"."FIT-506 LOW TIMER PV", DONE =>)
   END_RUNG
   RUNG wire#powerrail
      { S7_Templates := "SrcType := Int" } NE_Contact(in1 := "MODE SELECTION DB".EDI."PROCESS BUFF", in2 := 2)
   END_RUNG wire#w5
   RUNG wire#powerrail
      { S7_Templates := "SrcType := Int" } NE_Contact(in1 := "INTERLOCK DB"."EDI PARAMETER BUFF"."FIT-506 LOW / HIGH BUFF", in2 := 1)
   END_RUNG wire#w5
   RUNG wire#powerrail
      { S7_Templates := "SrcType := Int" } EQ_Contact(in1 := "MODE SELECTION DB".EDI."MODE BUFF", in2 := 1)
      { S7_Templates := "SrcType := Int" } EQ_Contact(in1 := "MODE SELECTION DB".EDI."PROCESS BUFF", in2 := 2)
      Contact( "EDI DB"."EDI FEED PUMP 401ABC" )
      { S7_Templates := "time_type := Time" } "IEC_Timer_0_DB_181".TON(pt := T#20S, et =>)
      { S7_Templates := "SrcType := Int" } EQ_Contact(in1 := "INTERLOCK DB"."EDI PARAMETER BUFF"."FIT-506 LOW / HIGH BUFF", in2 := 1)
      Contact( "PUMP SELECTION"."EDI-501" )
   END_RUNG wire#w6
   RUNG wire#powerrail
      "TIMING_SECS_DB_25"(RESET := wire#w7, INPUT := wire#w8, "SET TIME" := "INTERLOCK DB"."EDI SET TIMER"."FIT-506 HIGH TIMER SET", "PRESENT VALUE OF TIME" => "INTERLOCK DB"."EDI PV TIMER"."FIT-506 HIGH TIMER PV", DONE =>)
   END_RUNG
   RUNG wire#powerrail
      { S7_Templates := "SrcType := Int" } NE_Contact(in1 := "MODE SELECTION DB".EDI."PROCESS BUFF", in2 := 2)
   END_RUNG wire#w7
   RUNG wire#powerrail
      { S7_Templates := "SrcType := Int" } NE_Contact(in1 := "INTERLOCK DB"."EDI PARAMETER BUFF"."FIT-506 LOW / HIGH BUFF", in2 := 2)
   END_RUNG wire#w7
   RUNG wire#powerrail
      { S7_Templates := "SrcType := Int" } EQ_Contact(in1 := "MODE SELECTION DB".EDI."MODE BUFF", in2 := 1)
      { S7_Templates := "SrcType := Int" } EQ_Contact(in1 := "MODE SELECTION DB".EDI."PROCESS BUFF", in2 := 2)
      Contact( "EDI DB"."EDI FEED PUMP 401ABC" )
      { S7_Templates := "time_type := Time" } "IEC_Timer_0_DB_182".TON(pt := T#20S, et =>)
      { S7_Templates := "SrcType := Int" } EQ_Contact(in1 := "INTERLOCK DB"."EDI PARAMETER BUFF"."FIT-506 LOW / HIGH BUFF", in2 := 2)
      Contact( "PUMP SELECTION"."EDI-501" )
   END_RUNG wire#w8
   // the same network as SCL:
   #_w1 := "MODE SELECTION DB".EDI."MODE BUFF" = 1;
   "IEC_Timer_0_DB_198".TON(IN := #_w1 AND ("MODE SELECTION DB".EDI."PROCESS BUFF" = 2) AND "EDI DB"."EDI FEED PUMP 401ABC",
                           PT := T#15S);
   "IEC_Timer_0_DB_62".TON(IN := "IEC_Timer_0_DB_198".Q AND ("AI SCALING DB".PV."FLOW INDICATOR TRANSMITTER 506" < "INTERLOCK DB"."EDI SET PARAMETER"."FIT-506 LOW"),
                           PT := T#10S);
   IF "IEC_Timer_0_DB_62".Q THEN "INTERLOCK DB"."EDI PARAMETER BUFF"."FIT-506 LOW / HIGH BUFF" := 1; END_IF;
   "IEC_Timer_0_DB_63".TON(IN := "IEC_Timer_0_DB_198".Q AND ("AI SCALING DB".PV."FLOW INDICATOR TRANSMITTER 506" > "INTERLOCK DB"."EDI SET PARAMETER"."FIT-506 HIGH"),
                           PT := T#10S);
   IF "IEC_Timer_0_DB_63".Q THEN "INTERLOCK DB"."EDI PARAMETER BUFF"."FIT-506 LOW / HIGH BUFF" := 2; END_IF;
   IF #_w1 AND ((("AI SCALING DB".PV."FLOW INDICATOR TRANSMITTER 506" <= "INTERLOCK DB"."EDI SET PARAMETER"."FIT-506 HIGH") AND ("AI SCALING DB".PV."FLOW INDICATOR TRANSMITTER 506" >= "INTERLOCK DB"."EDI SET PARAMETER"."FIT-506 LOW")) OR NOT "EDI DB"."EDI FEED PUMP 401ABC") THEN
       "INTERLOCK DB"."EDI PARAMETER BUFF"."FIT-506 LOW / HIGH BUFF" := 0;
   END_IF;
   IF (("MODE SELECTION DB".EDI."MODE BUFF" = 1) AND ("MODE SELECTION DB".EDI."PROCESS BUFF" = 2) AND NOT "EDI DB"."EDI FEED PUMP 401ABC") OR ("MODE SELECTION DB".EDI."PROCESS BUFF" <> 2) THEN
       "INTERLOCK DB"."EDI PARAMETER BUFF"."FIT-506 LOW / HIGH BUFF" := 0;
   END_IF;
   "IEC_Timer_0_DB_181".TON(IN := ("MODE SELECTION DB".EDI."MODE BUFF" = 1) AND ("MODE SELECTION DB".EDI."PROCESS BUFF" = 2) AND "EDI DB"."EDI FEED PUMP 401ABC",
                           PT := T#20S);
   "TIMING_SECS_DB_24"("SET TIME" := "INTERLOCK DB"."EDI SET TIMER"."FIT-506 LOW TIMER SET",   // "TIMING_SECS"
                       RESET := ("MODE SELECTION DB".EDI."PROCESS BUFF" <> 2) OR ("INTERLOCK DB"."EDI PARAMETER BUFF"."FIT-506 LOW / HIGH BUFF" <> 1),
                       INPUT := "IEC_Timer_0_DB_181".Q AND ("INTERLOCK DB"."EDI PARAMETER BUFF"."FIT-506 LOW / HIGH BUFF" = 1) AND "PUMP SELECTION"."EDI-501",
                       "PRESENT VALUE OF TIME" => "INTERLOCK DB"."EDI PV TIMER"."FIT-506 LOW TIMER PV");
   "IEC_Timer_0_DB_182".TON(IN := ("MODE SELECTION DB".EDI."MODE BUFF" = 1) AND ("MODE SELECTION DB".EDI."PROCESS BUFF" = 2) AND "EDI DB"."EDI FEED PUMP 401ABC",
                           PT := T#20S);
   "TIMING_SECS_DB_25"("SET TIME" := "INTERLOCK DB"."EDI SET TIMER"."FIT-506 HIGH TIMER SET",   // "TIMING_SECS"
                       RESET := ("MODE SELECTION DB".EDI."PROCESS BUFF" <> 2) OR ("INTERLOCK DB"."EDI PARAMETER BUFF"."FIT-506 LOW / HIGH BUFF" <> 2),
                       INPUT := "IEC_Timer_0_DB_182".Q AND ("INTERLOCK DB"."EDI PARAMETER BUFF"."FIT-506 LOW / HIGH BUFF" = 2) AND "PUMP SELECTION"."EDI-501",
                       "PRESENT VALUE OF TIME" => "INTERLOCK DB"."EDI PV TIMER"."FIT-506 HIGH TIMER PV");
END_REGION

REGION Network 45: FIT-507 LOW / HIGH
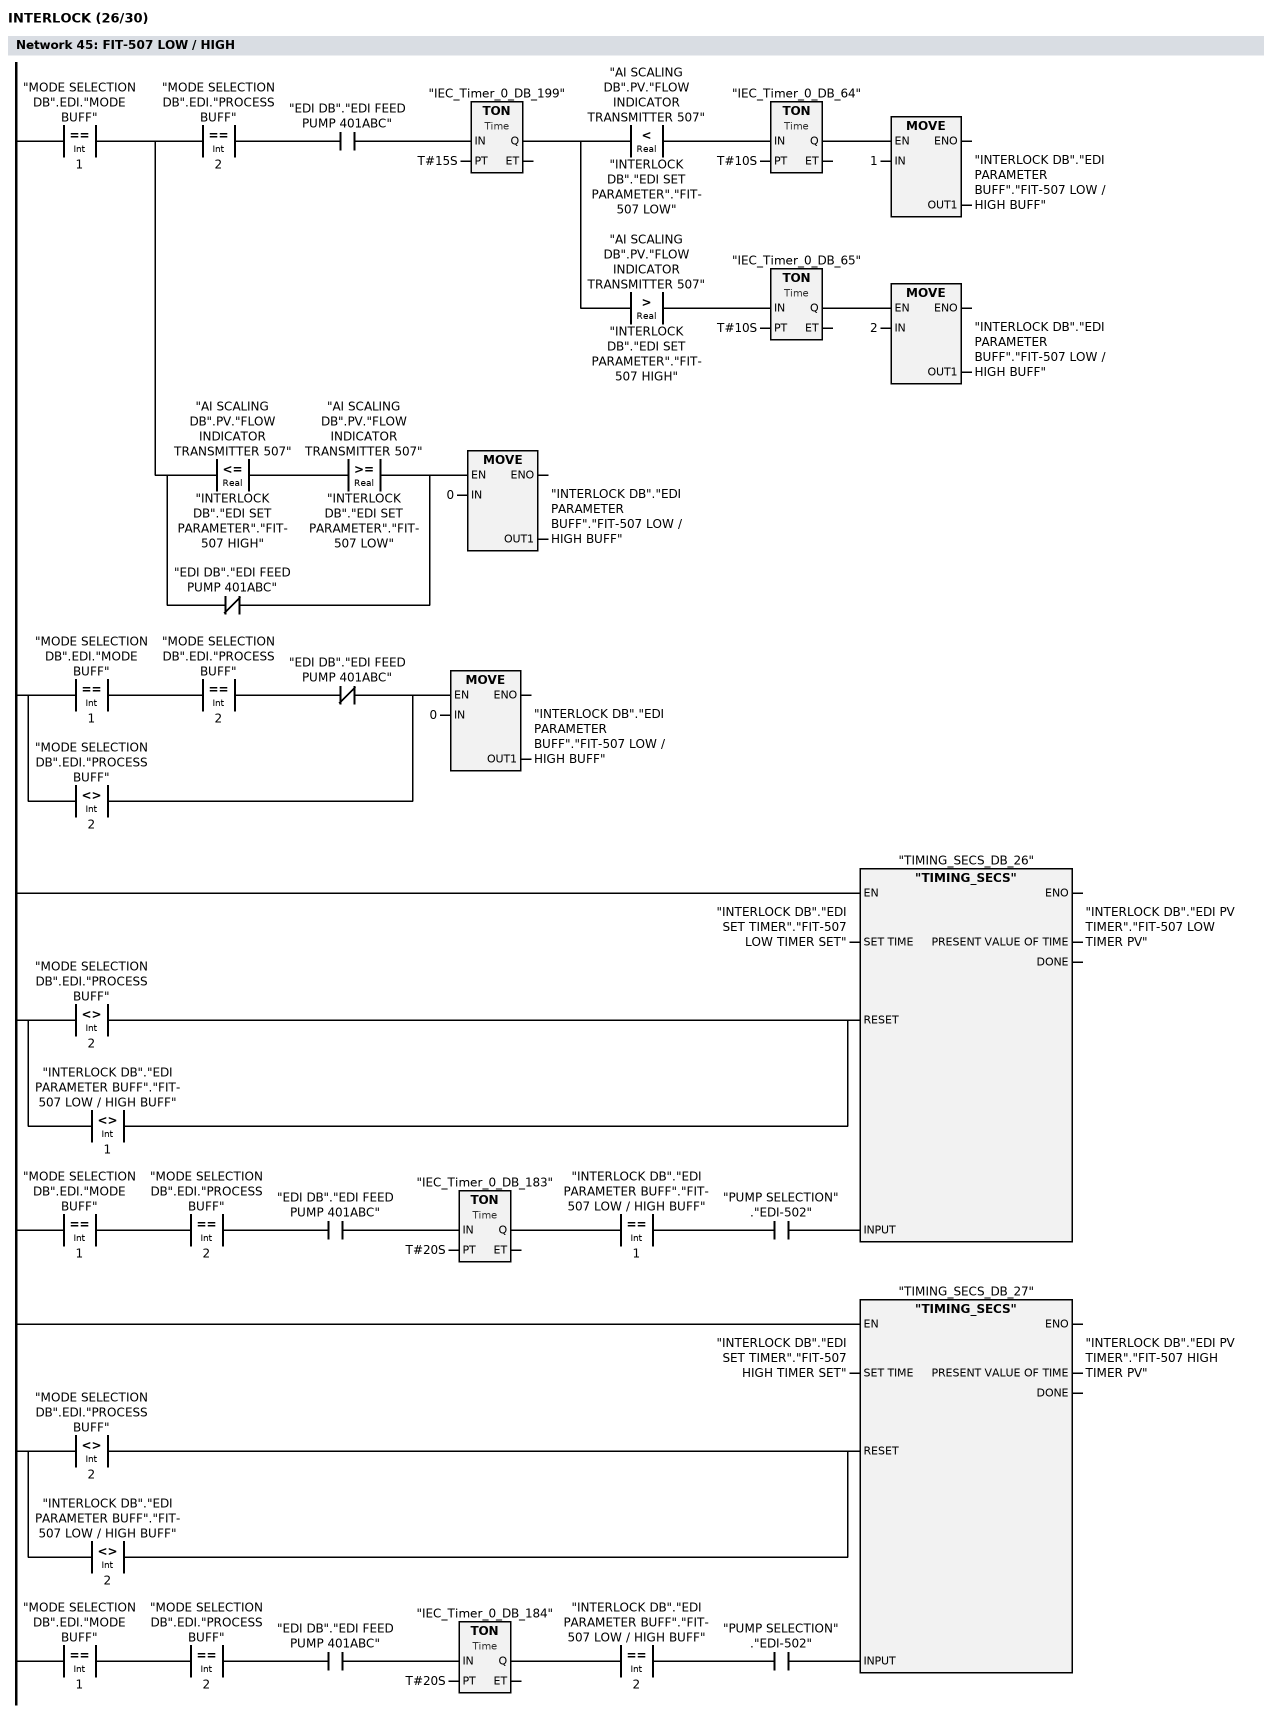
   RUNG wire#powerrail
      { S7_Templates := "SrcType := Int" } EQ_Contact(in1 := "MODE SELECTION DB".EDI."MODE BUFF", in2 := 1)
      wire#w1
      { S7_Templates := "SrcType := Int" } EQ_Contact(in1 := "MODE SELECTION DB".EDI."PROCESS BUFF", in2 := 2)
      Contact( "EDI DB"."EDI FEED PUMP 401ABC" )
      { S7_Templates := "time_type := Time" } "IEC_Timer_0_DB_199".TON(pt := T#15S, et =>)
      wire#w2
      { S7_Templates := "SrcType := Real" } LT_Contact(in1 := "AI SCALING DB".PV."FLOW INDICATOR TRANSMITTER 507", in2 := "INTERLOCK DB"."EDI SET PARAMETER"."FIT-507 LOW")
      { S7_Templates := "time_type := Time" } "IEC_Timer_0_DB_64".TON(pt := T#10S, et =>)
      Move(in := 1, out1 => "INTERLOCK DB"."EDI PARAMETER BUFF"."FIT-507 LOW / HIGH BUFF")
   END_RUNG
   RUNG wire#w2
      { S7_Templates := "SrcType := Real" } GT_Contact(in1 := "AI SCALING DB".PV."FLOW INDICATOR TRANSMITTER 507", in2 := "INTERLOCK DB"."EDI SET PARAMETER"."FIT-507 HIGH")
      { S7_Templates := "time_type := Time" } "IEC_Timer_0_DB_65".TON(pt := T#10S, et =>)
      Move(in := 2, out1 => "INTERLOCK DB"."EDI PARAMETER BUFF"."FIT-507 LOW / HIGH BUFF")
   END_RUNG
   RUNG wire#w1
      { S7_Templates := "SrcType := Real" } LE_Contact(in1 := "AI SCALING DB".PV."FLOW INDICATOR TRANSMITTER 507", in2 := "INTERLOCK DB"."EDI SET PARAMETER"."FIT-507 HIGH")
      { S7_Templates := "SrcType := Real" } GE_Contact(in1 := "AI SCALING DB".PV."FLOW INDICATOR TRANSMITTER 507", in2 := "INTERLOCK DB"."EDI SET PARAMETER"."FIT-507 LOW")
      wire#w3
      Move(in := 0, out1 => "INTERLOCK DB"."EDI PARAMETER BUFF"."FIT-507 LOW / HIGH BUFF")
   END_RUNG
   RUNG wire#w1
      I_Contact( "EDI DB"."EDI FEED PUMP 401ABC" )
   END_RUNG wire#w3
   RUNG wire#powerrail
      { S7_Templates := "SrcType := Int" } EQ_Contact(in1 := "MODE SELECTION DB".EDI."MODE BUFF", in2 := 1)
      { S7_Templates := "SrcType := Int" } EQ_Contact(in1 := "MODE SELECTION DB".EDI."PROCESS BUFF", in2 := 2)
      I_Contact( "EDI DB"."EDI FEED PUMP 401ABC" )
      wire#w4
      Move(in := 0, out1 => "INTERLOCK DB"."EDI PARAMETER BUFF"."FIT-507 LOW / HIGH BUFF")
   END_RUNG
   RUNG wire#powerrail
      { S7_Templates := "SrcType := Int" } NE_Contact(in1 := "MODE SELECTION DB".EDI."PROCESS BUFF", in2 := 2)
   END_RUNG wire#w4
   RUNG wire#powerrail
      "TIMING_SECS_DB_26"(RESET := wire#w5, INPUT := wire#w6, "SET TIME" := "INTERLOCK DB"."EDI SET TIMER"."FIT-507 LOW TIMER SET", "PRESENT VALUE OF TIME" => "INTERLOCK DB"."EDI PV TIMER"."FIT-507 LOW TIMER PV", DONE =>)
   END_RUNG
   RUNG wire#powerrail
      { S7_Templates := "SrcType := Int" } NE_Contact(in1 := "MODE SELECTION DB".EDI."PROCESS BUFF", in2 := 2)
   END_RUNG wire#w5
   RUNG wire#powerrail
      { S7_Templates := "SrcType := Int" } NE_Contact(in1 := "INTERLOCK DB"."EDI PARAMETER BUFF"."FIT-507 LOW / HIGH BUFF", in2 := 1)
   END_RUNG wire#w5
   RUNG wire#powerrail
      { S7_Templates := "SrcType := Int" } EQ_Contact(in1 := "MODE SELECTION DB".EDI."MODE BUFF", in2 := 1)
      { S7_Templates := "SrcType := Int" } EQ_Contact(in1 := "MODE SELECTION DB".EDI."PROCESS BUFF", in2 := 2)
      Contact( "EDI DB"."EDI FEED PUMP 401ABC" )
      { S7_Templates := "time_type := Time" } "IEC_Timer_0_DB_183".TON(pt := T#20S, et =>)
      { S7_Templates := "SrcType := Int" } EQ_Contact(in1 := "INTERLOCK DB"."EDI PARAMETER BUFF"."FIT-507 LOW / HIGH BUFF", in2 := 1)
      Contact( "PUMP SELECTION"."EDI-502" )
   END_RUNG wire#w6
   RUNG wire#powerrail
      "TIMING_SECS_DB_27"(RESET := wire#w7, INPUT := wire#w8, "SET TIME" := "INTERLOCK DB"."EDI SET TIMER"."FIT-507 HIGH TIMER SET", "PRESENT VALUE OF TIME" => "INTERLOCK DB"."EDI PV TIMER"."FIT-507 HIGH TIMER PV", DONE =>)
   END_RUNG
   RUNG wire#powerrail
      { S7_Templates := "SrcType := Int" } NE_Contact(in1 := "MODE SELECTION DB".EDI."PROCESS BUFF", in2 := 2)
   END_RUNG wire#w7
   RUNG wire#powerrail
      { S7_Templates := "SrcType := Int" } NE_Contact(in1 := "INTERLOCK DB"."EDI PARAMETER BUFF"."FIT-507 LOW / HIGH BUFF", in2 := 2)
   END_RUNG wire#w7
   RUNG wire#powerrail
      { S7_Templates := "SrcType := Int" } EQ_Contact(in1 := "MODE SELECTION DB".EDI."MODE BUFF", in2 := 1)
      { S7_Templates := "SrcType := Int" } EQ_Contact(in1 := "MODE SELECTION DB".EDI."PROCESS BUFF", in2 := 2)
      Contact( "EDI DB"."EDI FEED PUMP 401ABC" )
      { S7_Templates := "time_type := Time" } "IEC_Timer_0_DB_184".TON(pt := T#20S, et =>)
      { S7_Templates := "SrcType := Int" } EQ_Contact(in1 := "INTERLOCK DB"."EDI PARAMETER BUFF"."FIT-507 LOW / HIGH BUFF", in2 := 2)
      Contact( "PUMP SELECTION"."EDI-502" )
   END_RUNG wire#w8
   // the same network as SCL:
   #_w1 := "MODE SELECTION DB".EDI."MODE BUFF" = 1;
   "IEC_Timer_0_DB_199".TON(IN := #_w1 AND ("MODE SELECTION DB".EDI."PROCESS BUFF" = 2) AND "EDI DB"."EDI FEED PUMP 401ABC",
                           PT := T#15S);
   "IEC_Timer_0_DB_64".TON(IN := "IEC_Timer_0_DB_199".Q AND ("AI SCALING DB".PV."FLOW INDICATOR TRANSMITTER 507" < "INTERLOCK DB"."EDI SET PARAMETER"."FIT-507 LOW"),
                           PT := T#10S);
   IF "IEC_Timer_0_DB_64".Q THEN "INTERLOCK DB"."EDI PARAMETER BUFF"."FIT-507 LOW / HIGH BUFF" := 1; END_IF;
   "IEC_Timer_0_DB_65".TON(IN := "IEC_Timer_0_DB_199".Q AND ("AI SCALING DB".PV."FLOW INDICATOR TRANSMITTER 507" > "INTERLOCK DB"."EDI SET PARAMETER"."FIT-507 HIGH"),
                           PT := T#10S);
   IF "IEC_Timer_0_DB_65".Q THEN "INTERLOCK DB"."EDI PARAMETER BUFF"."FIT-507 LOW / HIGH BUFF" := 2; END_IF;
   IF #_w1 AND ((("AI SCALING DB".PV."FLOW INDICATOR TRANSMITTER 507" <= "INTERLOCK DB"."EDI SET PARAMETER"."FIT-507 HIGH") AND ("AI SCALING DB".PV."FLOW INDICATOR TRANSMITTER 507" >= "INTERLOCK DB"."EDI SET PARAMETER"."FIT-507 LOW")) OR NOT "EDI DB"."EDI FEED PUMP 401ABC") THEN
       "INTERLOCK DB"."EDI PARAMETER BUFF"."FIT-507 LOW / HIGH BUFF" := 0;
   END_IF;
   IF (("MODE SELECTION DB".EDI."MODE BUFF" = 1) AND ("MODE SELECTION DB".EDI."PROCESS BUFF" = 2) AND NOT "EDI DB"."EDI FEED PUMP 401ABC") OR ("MODE SELECTION DB".EDI."PROCESS BUFF" <> 2) THEN
       "INTERLOCK DB"."EDI PARAMETER BUFF"."FIT-507 LOW / HIGH BUFF" := 0;
   END_IF;
   "IEC_Timer_0_DB_183".TON(IN := ("MODE SELECTION DB".EDI."MODE BUFF" = 1) AND ("MODE SELECTION DB".EDI."PROCESS BUFF" = 2) AND "EDI DB"."EDI FEED PUMP 401ABC",
                           PT := T#20S);
   "TIMING_SECS_DB_26"("SET TIME" := "INTERLOCK DB"."EDI SET TIMER"."FIT-507 LOW TIMER SET",   // "TIMING_SECS"
                       RESET := ("MODE SELECTION DB".EDI."PROCESS BUFF" <> 2) OR ("INTERLOCK DB"."EDI PARAMETER BUFF"."FIT-507 LOW / HIGH BUFF" <> 1),
                       INPUT := "IEC_Timer_0_DB_183".Q AND ("INTERLOCK DB"."EDI PARAMETER BUFF"."FIT-507 LOW / HIGH BUFF" = 1) AND "PUMP SELECTION"."EDI-502",
                       "PRESENT VALUE OF TIME" => "INTERLOCK DB"."EDI PV TIMER"."FIT-507 LOW TIMER PV");
   "IEC_Timer_0_DB_184".TON(IN := ("MODE SELECTION DB".EDI."MODE BUFF" = 1) AND ("MODE SELECTION DB".EDI."PROCESS BUFF" = 2) AND "EDI DB"."EDI FEED PUMP 401ABC",
                           PT := T#20S);
   "TIMING_SECS_DB_27"("SET TIME" := "INTERLOCK DB"."EDI SET TIMER"."FIT-507 HIGH TIMER SET",   // "TIMING_SECS"
                       RESET := ("MODE SELECTION DB".EDI."PROCESS BUFF" <> 2) OR ("INTERLOCK DB"."EDI PARAMETER BUFF"."FIT-507 LOW / HIGH BUFF" <> 2),
                       INPUT := "IEC_Timer_0_DB_184".Q AND ("INTERLOCK DB"."EDI PARAMETER BUFF"."FIT-507 LOW / HIGH BUFF" = 2) AND "PUMP SELECTION"."EDI-502",
                       "PRESENT VALUE OF TIME" => "INTERLOCK DB"."EDI PV TIMER"."FIT-507 HIGH TIMER PV");
END_REGION

REGION Network 46: FIT-508 LOW / HIGH
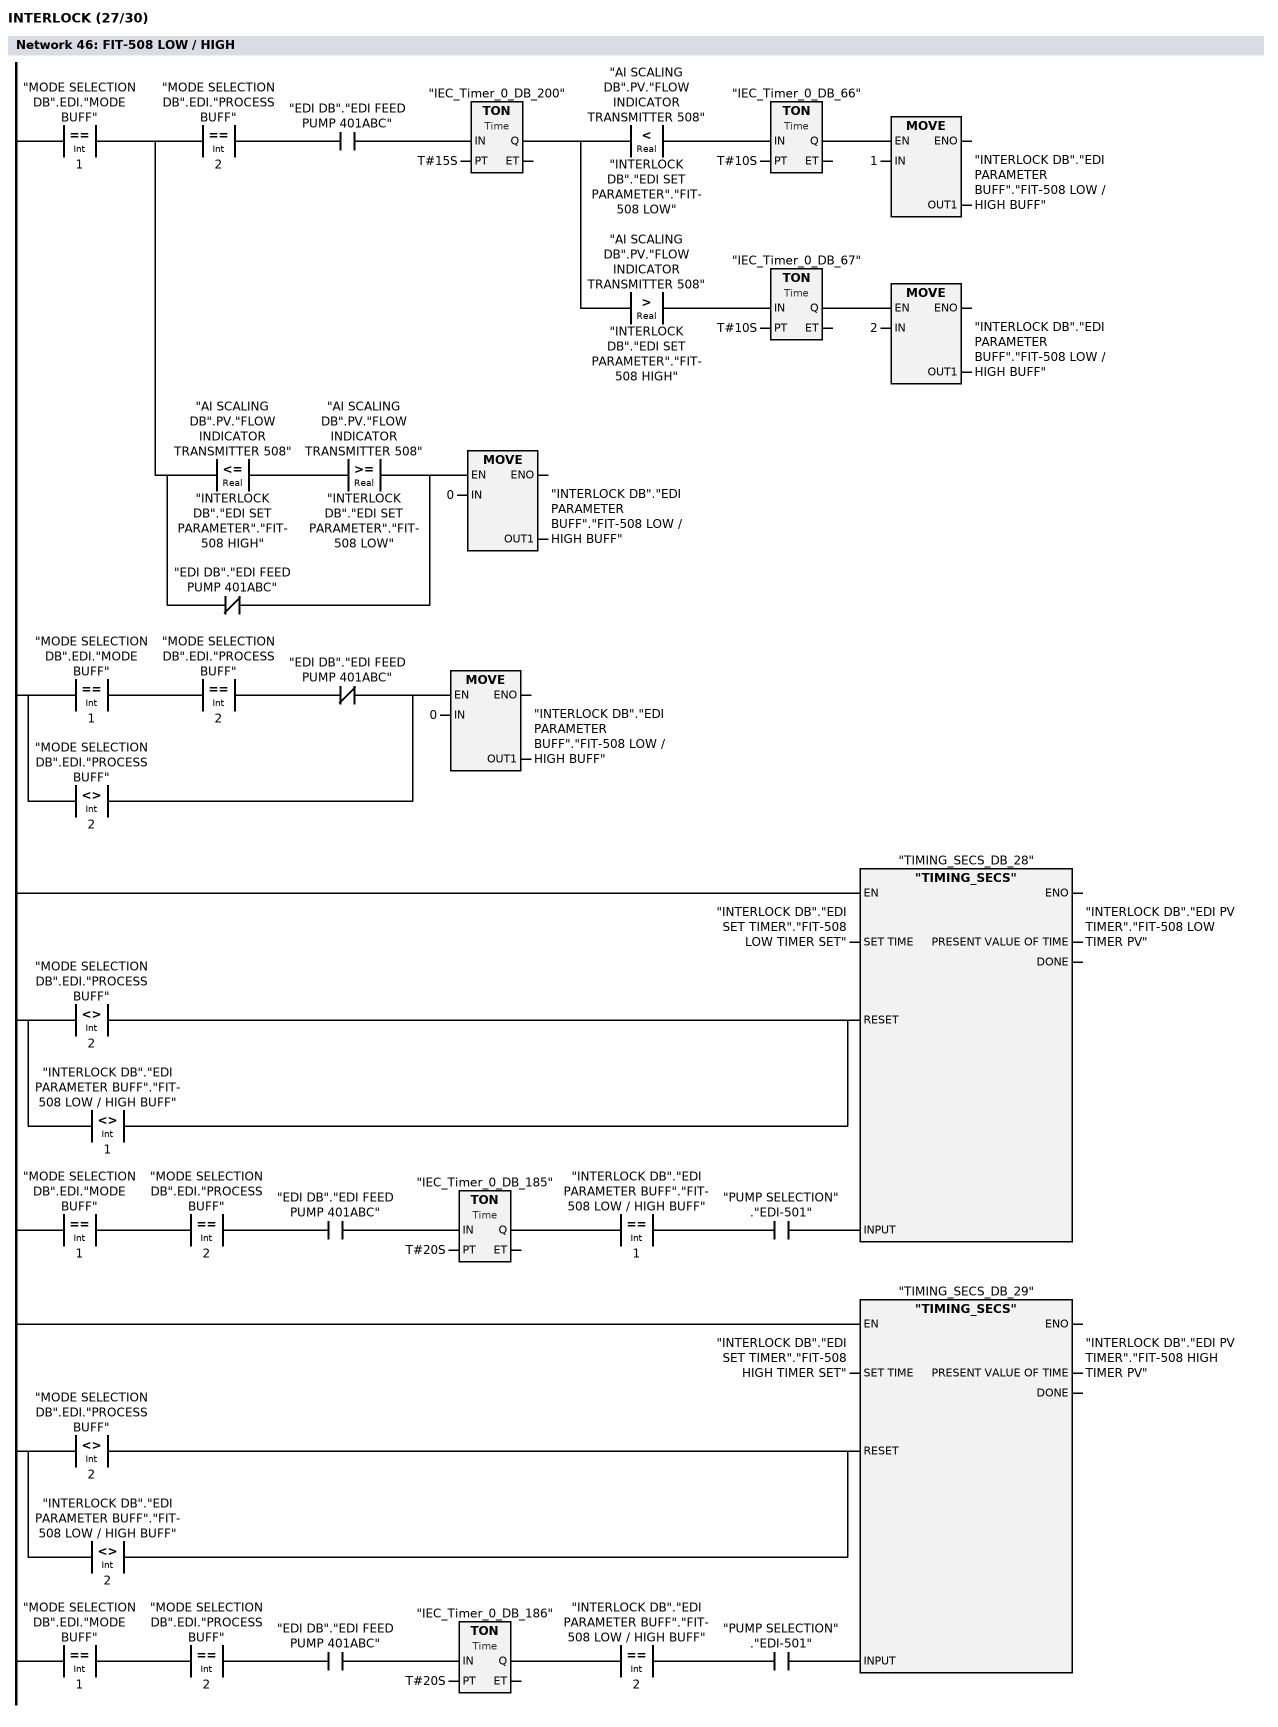
   RUNG wire#powerrail
      { S7_Templates := "SrcType := Int" } EQ_Contact(in1 := "MODE SELECTION DB".EDI."MODE BUFF", in2 := 1)
      wire#w1
      { S7_Templates := "SrcType := Int" } EQ_Contact(in1 := "MODE SELECTION DB".EDI."PROCESS BUFF", in2 := 2)
      Contact( "EDI DB"."EDI FEED PUMP 401ABC" )
      { S7_Templates := "time_type := Time" } "IEC_Timer_0_DB_200".TON(pt := T#15S, et =>)
      wire#w2
      { S7_Templates := "SrcType := Real" } LT_Contact(in1 := "AI SCALING DB".PV."FLOW INDICATOR TRANSMITTER 508", in2 := "INTERLOCK DB"."EDI SET PARAMETER"."FIT-508 LOW")
      { S7_Templates := "time_type := Time" } "IEC_Timer_0_DB_66".TON(pt := T#10S, et =>)
      Move(in := 1, out1 => "INTERLOCK DB"."EDI PARAMETER BUFF"."FIT-508 LOW / HIGH BUFF")
   END_RUNG
   RUNG wire#w2
      { S7_Templates := "SrcType := Real" } GT_Contact(in1 := "AI SCALING DB".PV."FLOW INDICATOR TRANSMITTER 508", in2 := "INTERLOCK DB"."EDI SET PARAMETER"."FIT-508 HIGH")
      { S7_Templates := "time_type := Time" } "IEC_Timer_0_DB_67".TON(pt := T#10S, et =>)
      Move(in := 2, out1 => "INTERLOCK DB"."EDI PARAMETER BUFF"."FIT-508 LOW / HIGH BUFF")
   END_RUNG
   RUNG wire#w1
      { S7_Templates := "SrcType := Real" } LE_Contact(in1 := "AI SCALING DB".PV."FLOW INDICATOR TRANSMITTER 508", in2 := "INTERLOCK DB"."EDI SET PARAMETER"."FIT-508 HIGH")
      { S7_Templates := "SrcType := Real" } GE_Contact(in1 := "AI SCALING DB".PV."FLOW INDICATOR TRANSMITTER 508", in2 := "INTERLOCK DB"."EDI SET PARAMETER"."FIT-508 LOW")
      wire#w3
      Move(in := 0, out1 => "INTERLOCK DB"."EDI PARAMETER BUFF"."FIT-508 LOW / HIGH BUFF")
   END_RUNG
   RUNG wire#w1
      I_Contact( "EDI DB"."EDI FEED PUMP 401ABC" )
   END_RUNG wire#w3
   RUNG wire#powerrail
      { S7_Templates := "SrcType := Int" } EQ_Contact(in1 := "MODE SELECTION DB".EDI."MODE BUFF", in2 := 1)
      { S7_Templates := "SrcType := Int" } EQ_Contact(in1 := "MODE SELECTION DB".EDI."PROCESS BUFF", in2 := 2)
      I_Contact( "EDI DB"."EDI FEED PUMP 401ABC" )
      wire#w4
      Move(in := 0, out1 => "INTERLOCK DB"."EDI PARAMETER BUFF"."FIT-508 LOW / HIGH BUFF")
   END_RUNG
   RUNG wire#powerrail
      { S7_Templates := "SrcType := Int" } NE_Contact(in1 := "MODE SELECTION DB".EDI."PROCESS BUFF", in2 := 2)
   END_RUNG wire#w4
   RUNG wire#powerrail
      "TIMING_SECS_DB_28"(RESET := wire#w5, INPUT := wire#w6, "SET TIME" := "INTERLOCK DB"."EDI SET TIMER"."FIT-508 LOW TIMER SET", "PRESENT VALUE OF TIME" => "INTERLOCK DB"."EDI PV TIMER"."FIT-508 LOW TIMER PV", DONE =>)
   END_RUNG
   RUNG wire#powerrail
      { S7_Templates := "SrcType := Int" } NE_Contact(in1 := "MODE SELECTION DB".EDI."PROCESS BUFF", in2 := 2)
   END_RUNG wire#w5
   RUNG wire#powerrail
      { S7_Templates := "SrcType := Int" } NE_Contact(in1 := "INTERLOCK DB"."EDI PARAMETER BUFF"."FIT-508 LOW / HIGH BUFF", in2 := 1)
   END_RUNG wire#w5
   RUNG wire#powerrail
      { S7_Templates := "SrcType := Int" } EQ_Contact(in1 := "MODE SELECTION DB".EDI."MODE BUFF", in2 := 1)
      { S7_Templates := "SrcType := Int" } EQ_Contact(in1 := "MODE SELECTION DB".EDI."PROCESS BUFF", in2 := 2)
      Contact( "EDI DB"."EDI FEED PUMP 401ABC" )
      { S7_Templates := "time_type := Time" } "IEC_Timer_0_DB_185".TON(pt := T#20S, et =>)
      { S7_Templates := "SrcType := Int" } EQ_Contact(in1 := "INTERLOCK DB"."EDI PARAMETER BUFF"."FIT-508 LOW / HIGH BUFF", in2 := 1)
      Contact( "PUMP SELECTION"."EDI-501" )
   END_RUNG wire#w6
   RUNG wire#powerrail
      "TIMING_SECS_DB_29"(RESET := wire#w7, INPUT := wire#w8, "SET TIME" := "INTERLOCK DB"."EDI SET TIMER"."FIT-508 HIGH TIMER SET", "PRESENT VALUE OF TIME" => "INTERLOCK DB"."EDI PV TIMER"."FIT-508 HIGH TIMER PV", DONE =>)
   END_RUNG
   RUNG wire#powerrail
      { S7_Templates := "SrcType := Int" } NE_Contact(in1 := "MODE SELECTION DB".EDI."PROCESS BUFF", in2 := 2)
   END_RUNG wire#w7
   RUNG wire#powerrail
      { S7_Templates := "SrcType := Int" } NE_Contact(in1 := "INTERLOCK DB"."EDI PARAMETER BUFF"."FIT-508 LOW / HIGH BUFF", in2 := 2)
   END_RUNG wire#w7
   RUNG wire#powerrail
      { S7_Templates := "SrcType := Int" } EQ_Contact(in1 := "MODE SELECTION DB".EDI."MODE BUFF", in2 := 1)
      { S7_Templates := "SrcType := Int" } EQ_Contact(in1 := "MODE SELECTION DB".EDI."PROCESS BUFF", in2 := 2)
      Contact( "EDI DB"."EDI FEED PUMP 401ABC" )
      { S7_Templates := "time_type := Time" } "IEC_Timer_0_DB_186".TON(pt := T#20S, et =>)
      { S7_Templates := "SrcType := Int" } EQ_Contact(in1 := "INTERLOCK DB"."EDI PARAMETER BUFF"."FIT-508 LOW / HIGH BUFF", in2 := 2)
      Contact( "PUMP SELECTION"."EDI-501" )
   END_RUNG wire#w8
   // the same network as SCL:
   #_w1 := "MODE SELECTION DB".EDI."MODE BUFF" = 1;
   "IEC_Timer_0_DB_200".TON(IN := #_w1 AND ("MODE SELECTION DB".EDI."PROCESS BUFF" = 2) AND "EDI DB"."EDI FEED PUMP 401ABC",
                           PT := T#15S);
   "IEC_Timer_0_DB_66".TON(IN := "IEC_Timer_0_DB_200".Q AND ("AI SCALING DB".PV."FLOW INDICATOR TRANSMITTER 508" < "INTERLOCK DB"."EDI SET PARAMETER"."FIT-508 LOW"),
                           PT := T#10S);
   IF "IEC_Timer_0_DB_66".Q THEN "INTERLOCK DB"."EDI PARAMETER BUFF"."FIT-508 LOW / HIGH BUFF" := 1; END_IF;
   "IEC_Timer_0_DB_67".TON(IN := "IEC_Timer_0_DB_200".Q AND ("AI SCALING DB".PV."FLOW INDICATOR TRANSMITTER 508" > "INTERLOCK DB"."EDI SET PARAMETER"."FIT-508 HIGH"),
                           PT := T#10S);
   IF "IEC_Timer_0_DB_67".Q THEN "INTERLOCK DB"."EDI PARAMETER BUFF"."FIT-508 LOW / HIGH BUFF" := 2; END_IF;
   IF #_w1 AND ((("AI SCALING DB".PV."FLOW INDICATOR TRANSMITTER 508" <= "INTERLOCK DB"."EDI SET PARAMETER"."FIT-508 HIGH") AND ("AI SCALING DB".PV."FLOW INDICATOR TRANSMITTER 508" >= "INTERLOCK DB"."EDI SET PARAMETER"."FIT-508 LOW")) OR NOT "EDI DB"."EDI FEED PUMP 401ABC") THEN
       "INTERLOCK DB"."EDI PARAMETER BUFF"."FIT-508 LOW / HIGH BUFF" := 0;
   END_IF;
   IF (("MODE SELECTION DB".EDI."MODE BUFF" = 1) AND ("MODE SELECTION DB".EDI."PROCESS BUFF" = 2) AND NOT "EDI DB"."EDI FEED PUMP 401ABC") OR ("MODE SELECTION DB".EDI."PROCESS BUFF" <> 2) THEN
       "INTERLOCK DB"."EDI PARAMETER BUFF"."FIT-508 LOW / HIGH BUFF" := 0;
   END_IF;
   "IEC_Timer_0_DB_185".TON(IN := ("MODE SELECTION DB".EDI."MODE BUFF" = 1) AND ("MODE SELECTION DB".EDI."PROCESS BUFF" = 2) AND "EDI DB"."EDI FEED PUMP 401ABC",
                           PT := T#20S);
   "TIMING_SECS_DB_28"("SET TIME" := "INTERLOCK DB"."EDI SET TIMER"."FIT-508 LOW TIMER SET",   // "TIMING_SECS"
                       RESET := ("MODE SELECTION DB".EDI."PROCESS BUFF" <> 2) OR ("INTERLOCK DB"."EDI PARAMETER BUFF"."FIT-508 LOW / HIGH BUFF" <> 1),
                       INPUT := "IEC_Timer_0_DB_185".Q AND ("INTERLOCK DB"."EDI PARAMETER BUFF"."FIT-508 LOW / HIGH BUFF" = 1) AND "PUMP SELECTION"."EDI-501",
                       "PRESENT VALUE OF TIME" => "INTERLOCK DB"."EDI PV TIMER"."FIT-508 LOW TIMER PV");
   "IEC_Timer_0_DB_186".TON(IN := ("MODE SELECTION DB".EDI."MODE BUFF" = 1) AND ("MODE SELECTION DB".EDI."PROCESS BUFF" = 2) AND "EDI DB"."EDI FEED PUMP 401ABC",
                           PT := T#20S);
   "TIMING_SECS_DB_29"("SET TIME" := "INTERLOCK DB"."EDI SET TIMER"."FIT-508 HIGH TIMER SET",   // "TIMING_SECS"
                       RESET := ("MODE SELECTION DB".EDI."PROCESS BUFF" <> 2) OR ("INTERLOCK DB"."EDI PARAMETER BUFF"."FIT-508 LOW / HIGH BUFF" <> 2),
                       INPUT := "IEC_Timer_0_DB_186".Q AND ("INTERLOCK DB"."EDI PARAMETER BUFF"."FIT-508 LOW / HIGH BUFF" = 2) AND "PUMP SELECTION"."EDI-501",
                       "PRESENT VALUE OF TIME" => "INTERLOCK DB"."EDI PV TIMER"."FIT-508 HIGH TIMER PV");
END_REGION

REGION Network 47: pH-501 - LOW / High
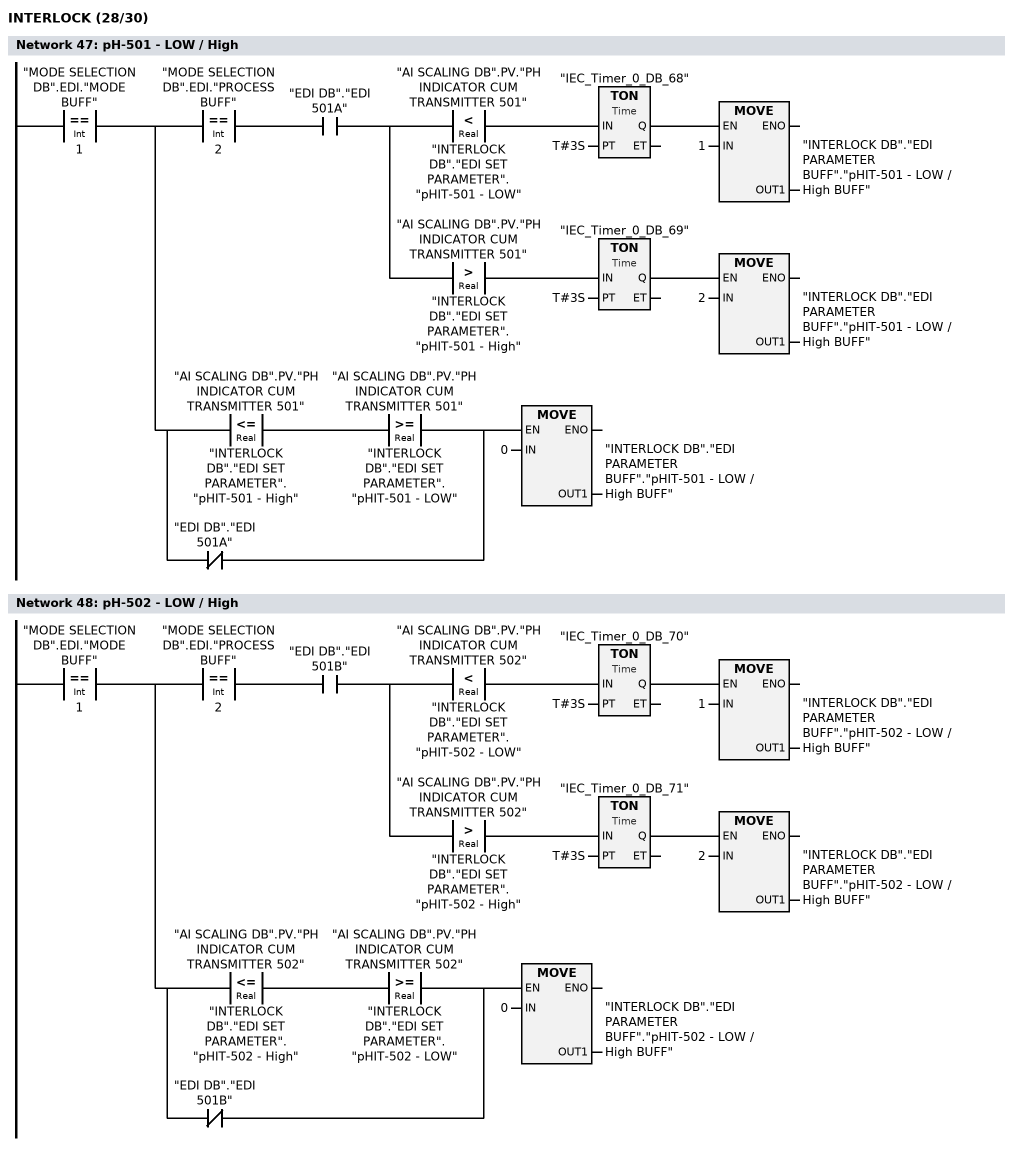
   RUNG wire#powerrail
      { S7_Templates := "SrcType := Int" } EQ_Contact(in1 := "MODE SELECTION DB".EDI."MODE BUFF", in2 := 1)
      wire#w1
      { S7_Templates := "SrcType := Int" } EQ_Contact(in1 := "MODE SELECTION DB".EDI."PROCESS BUFF", in2 := 2)
      Contact( "EDI DB"."EDI 501A" )
      wire#w2
      { S7_Templates := "SrcType := Real" } LT_Contact(in1 := "AI SCALING DB".PV."PH INDICATOR CUM TRANSMITTER 501", in2 := "INTERLOCK DB"."EDI SET PARAMETER"."pHIT-501 - LOW")
      { S7_Templates := "time_type := Time" } "IEC_Timer_0_DB_68".TON(pt := T#3S, et =>)
      Move(in := 1, out1 => "INTERLOCK DB"."EDI PARAMETER BUFF"."pHIT-501 - LOW / High BUFF")
   END_RUNG
   RUNG wire#w2
      { S7_Templates := "SrcType := Real" } GT_Contact(in1 := "AI SCALING DB".PV."PH INDICATOR CUM TRANSMITTER 501", in2 := "INTERLOCK DB"."EDI SET PARAMETER"."pHIT-501 - High")
      { S7_Templates := "time_type := Time" } "IEC_Timer_0_DB_69".TON(pt := T#3S, et =>)
      Move(in := 2, out1 => "INTERLOCK DB"."EDI PARAMETER BUFF"."pHIT-501 - LOW / High BUFF")
   END_RUNG
   RUNG wire#w1
      { S7_Templates := "SrcType := Real" } LE_Contact(in1 := "AI SCALING DB".PV."PH INDICATOR CUM TRANSMITTER 501", in2 := "INTERLOCK DB"."EDI SET PARAMETER"."pHIT-501 - High")
      { S7_Templates := "SrcType := Real" } GE_Contact(in1 := "AI SCALING DB".PV."PH INDICATOR CUM TRANSMITTER 501", in2 := "INTERLOCK DB"."EDI SET PARAMETER"."pHIT-501 - LOW")
      wire#w3
      Move(in := 0, out1 => "INTERLOCK DB"."EDI PARAMETER BUFF"."pHIT-501 - LOW / High BUFF")
   END_RUNG
   RUNG wire#w1
      I_Contact( "EDI DB"."EDI 501A" )
   END_RUNG wire#w3
   // the same network as SCL:
   #_w1 := "MODE SELECTION DB".EDI."MODE BUFF" = 1;
   #_w2 := #_w1 AND ("MODE SELECTION DB".EDI."PROCESS BUFF" = 2) AND "EDI DB"."EDI 501A";
   "IEC_Timer_0_DB_68".TON(IN := #_w2 AND ("AI SCALING DB".PV."PH INDICATOR CUM TRANSMITTER 501" < "INTERLOCK DB"."EDI SET PARAMETER"."pHIT-501 - LOW"),
                           PT := T#3S);
   IF "IEC_Timer_0_DB_68".Q THEN
       "INTERLOCK DB"."EDI PARAMETER BUFF"."pHIT-501 - LOW / High BUFF" := 1;
   END_IF;
   "IEC_Timer_0_DB_69".TON(IN := #_w2 AND ("AI SCALING DB".PV."PH INDICATOR CUM TRANSMITTER 501" > "INTERLOCK DB"."EDI SET PARAMETER"."pHIT-501 - High"),
                           PT := T#3S);
   IF "IEC_Timer_0_DB_69".Q THEN
       "INTERLOCK DB"."EDI PARAMETER BUFF"."pHIT-501 - LOW / High BUFF" := 2;
   END_IF;
   IF #_w1 AND ((("AI SCALING DB".PV."PH INDICATOR CUM TRANSMITTER 501" <= "INTERLOCK DB"."EDI SET PARAMETER"."pHIT-501 - High") AND ("AI SCALING DB".PV."PH INDICATOR CUM TRANSMITTER 501" >= "INTERLOCK DB"."EDI SET PARAMETER"."pHIT-501 - LOW")) OR NOT "EDI DB"."EDI 501A") THEN
       "INTERLOCK DB"."EDI PARAMETER BUFF"."pHIT-501 - LOW / High BUFF" := 0;
   END_IF;
END_REGION

REGION Network 48: pH-502 - LOW / High
   RUNG wire#powerrail
      { S7_Templates := "SrcType := Int" } EQ_Contact(in1 := "MODE SELECTION DB".EDI."MODE BUFF", in2 := 1)
      wire#w1
      { S7_Templates := "SrcType := Int" } EQ_Contact(in1 := "MODE SELECTION DB".EDI."PROCESS BUFF", in2 := 2)
      Contact( "EDI DB"."EDI 501B" )
      wire#w2
      { S7_Templates := "SrcType := Real" } LT_Contact(in1 := "AI SCALING DB".PV."PH INDICATOR CUM TRANSMITTER 502", in2 := "INTERLOCK DB"."EDI SET PARAMETER"."pHIT-502 - LOW")
      { S7_Templates := "time_type := Time" } "IEC_Timer_0_DB_70".TON(pt := T#3S, et =>)
      Move(in := 1, out1 => "INTERLOCK DB"."EDI PARAMETER BUFF"."pHIT-502 - LOW / High BUFF")
   END_RUNG
   RUNG wire#w2
      { S7_Templates := "SrcType := Real" } GT_Contact(in1 := "AI SCALING DB".PV."PH INDICATOR CUM TRANSMITTER 502", in2 := "INTERLOCK DB"."EDI SET PARAMETER"."pHIT-502 - High")
      { S7_Templates := "time_type := Time" } "IEC_Timer_0_DB_71".TON(pt := T#3S, et =>)
      Move(in := 2, out1 => "INTERLOCK DB"."EDI PARAMETER BUFF"."pHIT-502 - LOW / High BUFF")
   END_RUNG
   RUNG wire#w1
      { S7_Templates := "SrcType := Real" } LE_Contact(in1 := "AI SCALING DB".PV."PH INDICATOR CUM TRANSMITTER 502", in2 := "INTERLOCK DB"."EDI SET PARAMETER"."pHIT-502 - High")
      { S7_Templates := "SrcType := Real" } GE_Contact(in1 := "AI SCALING DB".PV."PH INDICATOR CUM TRANSMITTER 502", in2 := "INTERLOCK DB"."EDI SET PARAMETER"."pHIT-502 - LOW")
      wire#w3
      Move(in := 0, out1 => "INTERLOCK DB"."EDI PARAMETER BUFF"."pHIT-502 - LOW / High BUFF")
   END_RUNG
   RUNG wire#w1
      I_Contact( "EDI DB"."EDI 501B" )
   END_RUNG wire#w3
   // the same network as SCL:
   #_w1 := "MODE SELECTION DB".EDI."MODE BUFF" = 1;
   #_w2 := #_w1 AND ("MODE SELECTION DB".EDI."PROCESS BUFF" = 2) AND "EDI DB"."EDI 501B";
   "IEC_Timer_0_DB_70".TON(IN := #_w2 AND ("AI SCALING DB".PV."PH INDICATOR CUM TRANSMITTER 502" < "INTERLOCK DB"."EDI SET PARAMETER"."pHIT-502 - LOW"),
                           PT := T#3S);
   IF "IEC_Timer_0_DB_70".Q THEN
       "INTERLOCK DB"."EDI PARAMETER BUFF"."pHIT-502 - LOW / High BUFF" := 1;
   END_IF;
   "IEC_Timer_0_DB_71".TON(IN := #_w2 AND ("AI SCALING DB".PV."PH INDICATOR CUM TRANSMITTER 502" > "INTERLOCK DB"."EDI SET PARAMETER"."pHIT-502 - High"),
                           PT := T#3S);
   IF "IEC_Timer_0_DB_71".Q THEN
       "INTERLOCK DB"."EDI PARAMETER BUFF"."pHIT-502 - LOW / High BUFF" := 2;
   END_IF;
   IF #_w1 AND ((("AI SCALING DB".PV."PH INDICATOR CUM TRANSMITTER 502" <= "INTERLOCK DB"."EDI SET PARAMETER"."pHIT-502 - High") AND ("AI SCALING DB".PV."PH INDICATOR CUM TRANSMITTER 502" >= "INTERLOCK DB"."EDI SET PARAMETER"."pHIT-502 - LOW")) OR NOT "EDI DB"."EDI 501B") THEN
       "INTERLOCK DB"."EDI PARAMETER BUFF"."pHIT-502 - LOW / High BUFF" := 0;
   END_IF;
END_REGION

REGION Network 49: RIT-501 HIGH
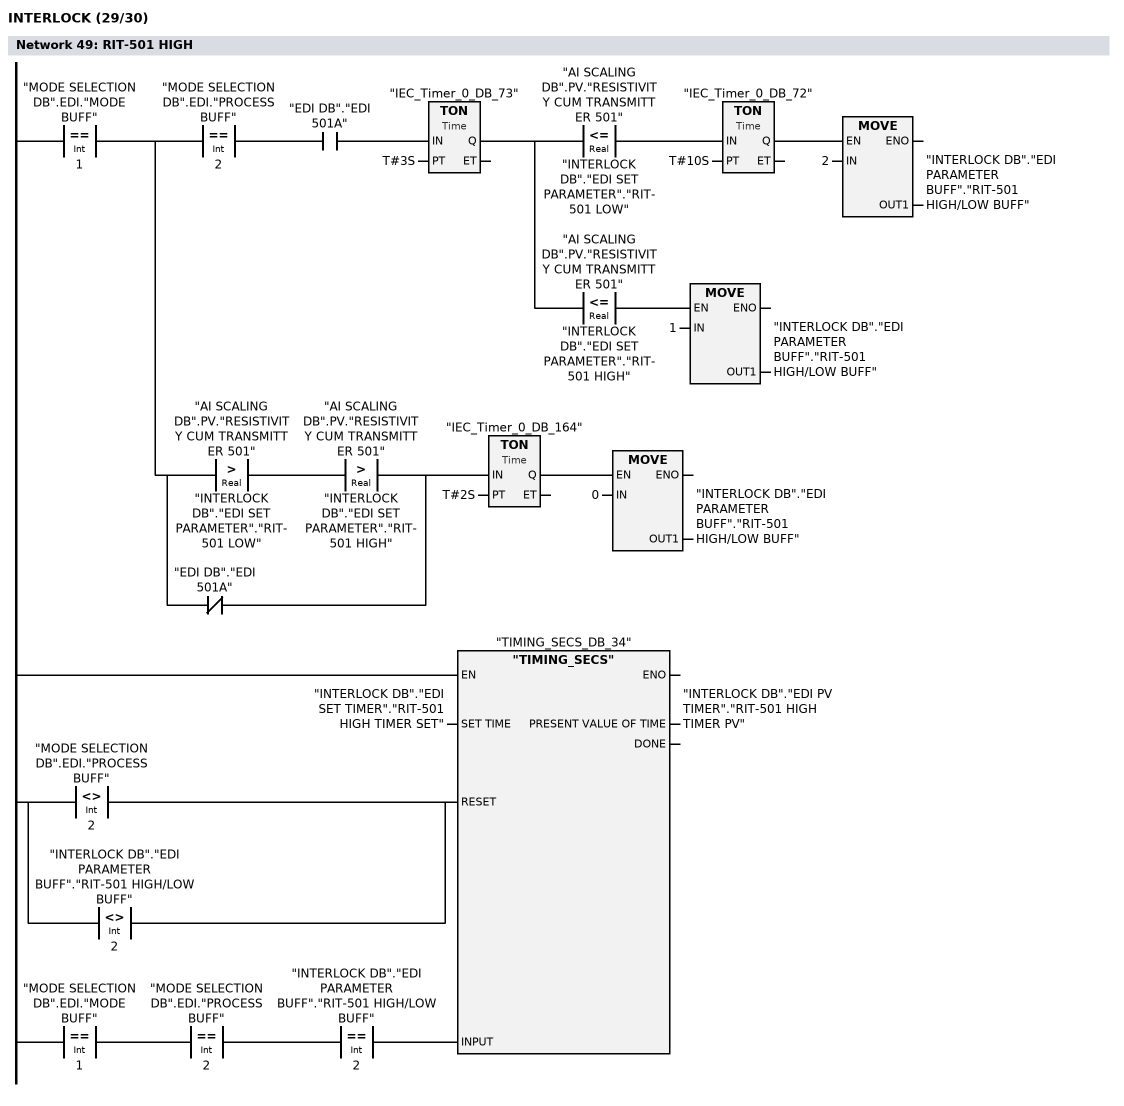
   RUNG wire#powerrail
      { S7_Templates := "SrcType := Int" } EQ_Contact(in1 := "MODE SELECTION DB".EDI."MODE BUFF", in2 := 1)
      wire#w1
      { S7_Templates := "SrcType := Int" } EQ_Contact(in1 := "MODE SELECTION DB".EDI."PROCESS BUFF", in2 := 2)
      Contact( "EDI DB"."EDI 501A" )
      { S7_Templates := "time_type := Time" } "IEC_Timer_0_DB_73".TON(pt := T#3S, et =>)
      wire#w2
      { S7_Templates := "SrcType := Real" } LE_Contact(in1 := "AI SCALING DB".PV."RESISTIVITY CUM TRANSMITTER 501", in2 := "INTERLOCK DB"."EDI SET PARAMETER"."RIT-501 LOW")
      { S7_Templates := "time_type := Time" } "IEC_Timer_0_DB_72".TON(pt := T#10S, et =>)
      Move(in := 2, out1 => "INTERLOCK DB"."EDI PARAMETER BUFF"."RIT-501 HIGH/LOW BUFF")
   END_RUNG
   RUNG wire#w2
      { S7_Templates := "SrcType := Real" } LE_Contact(in1 := "AI SCALING DB".PV."RESISTIVITY CUM TRANSMITTER 501", in2 := "INTERLOCK DB"."EDI SET PARAMETER"."RIT-501 HIGH")
      Move(in := 1, out1 => "INTERLOCK DB"."EDI PARAMETER BUFF"."RIT-501 HIGH/LOW BUFF")
   END_RUNG
   RUNG wire#w1
      { S7_Templates := "SrcType := Real" } GT_Contact(in1 := "AI SCALING DB".PV."RESISTIVITY CUM TRANSMITTER 501", in2 := "INTERLOCK DB"."EDI SET PARAMETER"."RIT-501 LOW")
      { S7_Templates := "SrcType := Real" } GT_Contact(in1 := "AI SCALING DB".PV."RESISTIVITY CUM TRANSMITTER 501", in2 := "INTERLOCK DB"."EDI SET PARAMETER"."RIT-501 HIGH")
      wire#w3
      { S7_Templates := "time_type := Time" } "IEC_Timer_0_DB_164".TON(pt := T#2S, et =>)
      Move(in := 0, out1 => "INTERLOCK DB"."EDI PARAMETER BUFF"."RIT-501 HIGH/LOW BUFF")
   END_RUNG
   RUNG wire#w1
      I_Contact( "EDI DB"."EDI 501A" )
   END_RUNG wire#w3
   RUNG wire#powerrail
      "TIMING_SECS_DB_34"(RESET := wire#w4, INPUT := wire#w5, "SET TIME" := "INTERLOCK DB"."EDI SET TIMER"."RIT-501 HIGH TIMER SET", "PRESENT VALUE OF TIME" => "INTERLOCK DB"."EDI PV TIMER"."RIT-501 HIGH TIMER PV", DONE =>)
   END_RUNG
   RUNG wire#powerrail
      { S7_Templates := "SrcType := Int" } NE_Contact(in1 := "MODE SELECTION DB".EDI."PROCESS BUFF", in2 := 2)
   END_RUNG wire#w4
   RUNG wire#powerrail
      { S7_Templates := "SrcType := Int" } NE_Contact(in1 := "INTERLOCK DB"."EDI PARAMETER BUFF"."RIT-501 HIGH/LOW BUFF", in2 := 2)
   END_RUNG wire#w4
   RUNG wire#powerrail
      { S7_Templates := "SrcType := Int" } EQ_Contact(in1 := "MODE SELECTION DB".EDI."MODE BUFF", in2 := 1)
      { S7_Templates := "SrcType := Int" } EQ_Contact(in1 := "MODE SELECTION DB".EDI."PROCESS BUFF", in2 := 2)
      { S7_Templates := "SrcType := Int" } EQ_Contact(in1 := "INTERLOCK DB"."EDI PARAMETER BUFF"."RIT-501 HIGH/LOW BUFF", in2 := 2)
   END_RUNG wire#w5
   // the same network as SCL:
   #_w1 := "MODE SELECTION DB".EDI."MODE BUFF" = 1;
   "IEC_Timer_0_DB_73".TON(IN := #_w1 AND ("MODE SELECTION DB".EDI."PROCESS BUFF" = 2) AND "EDI DB"."EDI 501A",
                           PT := T#3S);
   "IEC_Timer_0_DB_72".TON(IN := "IEC_Timer_0_DB_73".Q AND ("AI SCALING DB".PV."RESISTIVITY CUM TRANSMITTER 501" <= "INTERLOCK DB"."EDI SET PARAMETER"."RIT-501 LOW"),
                           PT := T#10S);
   IF "IEC_Timer_0_DB_72".Q THEN "INTERLOCK DB"."EDI PARAMETER BUFF"."RIT-501 HIGH/LOW BUFF" := 2; END_IF;
   IF "IEC_Timer_0_DB_73".Q AND ("AI SCALING DB".PV."RESISTIVITY CUM TRANSMITTER 501" <= "INTERLOCK DB"."EDI SET PARAMETER"."RIT-501 HIGH") THEN
       "INTERLOCK DB"."EDI PARAMETER BUFF"."RIT-501 HIGH/LOW BUFF" := 1;
   END_IF;
   "IEC_Timer_0_DB_164".TON(IN := #_w1 AND ((("AI SCALING DB".PV."RESISTIVITY CUM TRANSMITTER 501" > "INTERLOCK DB"."EDI SET PARAMETER"."RIT-501 LOW") AND ("AI SCALING DB".PV."RESISTIVITY CUM TRANSMITTER 501" > "INTERLOCK DB"."EDI SET PARAMETER"."RIT-501 HIGH")) OR NOT "EDI DB"."EDI 501A"),
                           PT := T#2S);
   IF "IEC_Timer_0_DB_164".Q THEN "INTERLOCK DB"."EDI PARAMETER BUFF"."RIT-501 HIGH/LOW BUFF" := 0; END_IF;
   "TIMING_SECS_DB_34"("SET TIME" := "INTERLOCK DB"."EDI SET TIMER"."RIT-501 HIGH TIMER SET",   // "TIMING_SECS"
                       RESET := ("MODE SELECTION DB".EDI."PROCESS BUFF" <> 2) OR ("INTERLOCK DB"."EDI PARAMETER BUFF"."RIT-501 HIGH/LOW BUFF" <> 2),
                       INPUT := ("MODE SELECTION DB".EDI."MODE BUFF" = 1) AND ("MODE SELECTION DB".EDI."PROCESS BUFF" = 2) AND ("INTERLOCK DB"."EDI PARAMETER BUFF"."RIT-501 HIGH/LOW BUFF" = 2),
                       "PRESENT VALUE OF TIME" => "INTERLOCK DB"."EDI PV TIMER"."RIT-501 HIGH TIMER PV");
END_REGION

REGION Network 50: RIT-502 HIGH
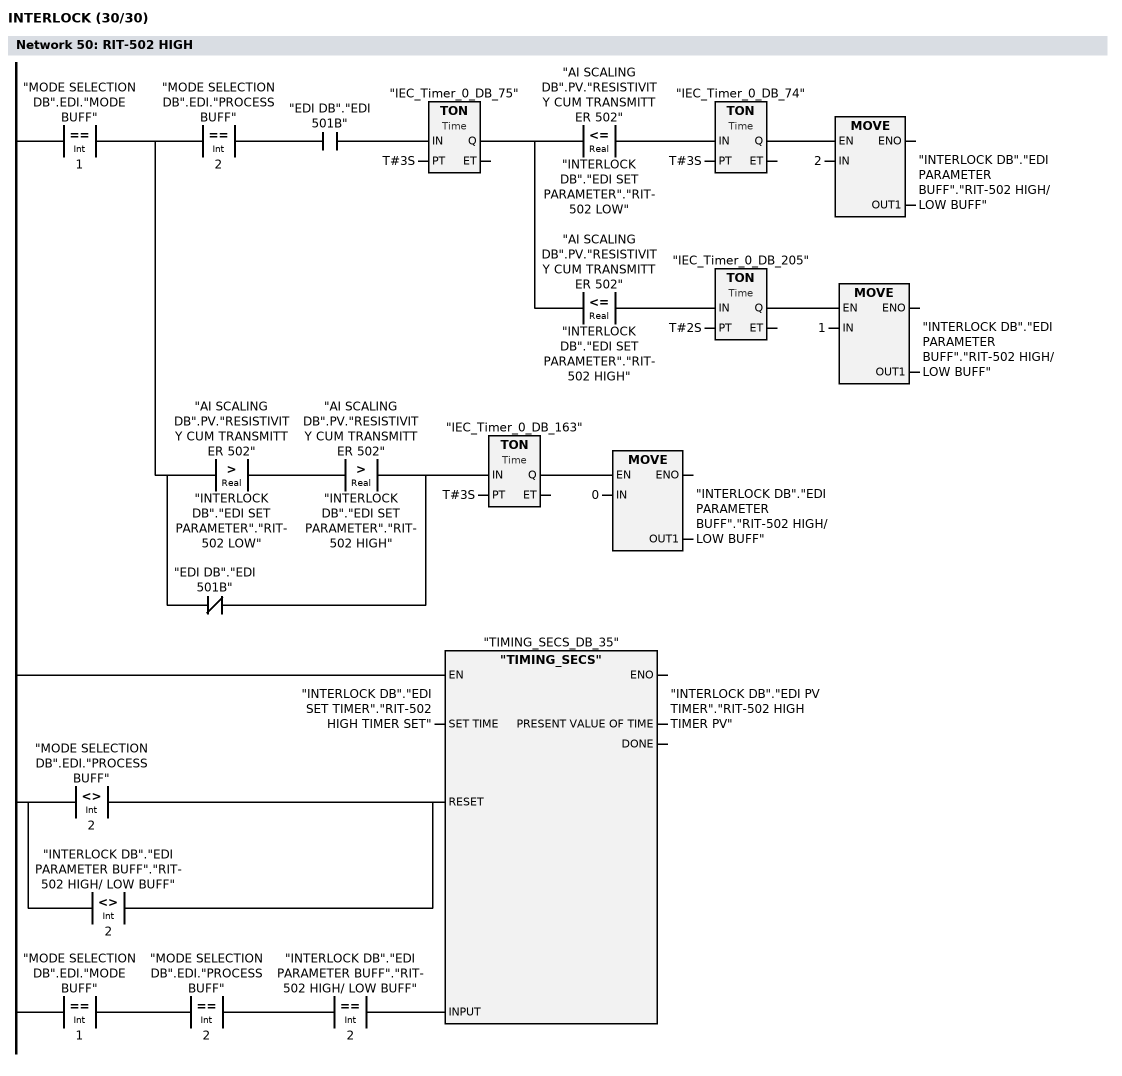
   RUNG wire#powerrail
      { S7_Templates := "SrcType := Int" } EQ_Contact(in1 := "MODE SELECTION DB".EDI."MODE BUFF", in2 := 1)
      wire#w1
      { S7_Templates := "SrcType := Int" } EQ_Contact(in1 := "MODE SELECTION DB".EDI."PROCESS BUFF", in2 := 2)
      Contact( "EDI DB"."EDI 501B" )
      { S7_Templates := "time_type := Time" } "IEC_Timer_0_DB_75".TON(pt := T#3S, et =>)
      wire#w2
      { S7_Templates := "SrcType := Real" } LE_Contact(in1 := "AI SCALING DB".PV."RESISTIVITY CUM TRANSMITTER 502", in2 := "INTERLOCK DB"."EDI SET PARAMETER"."RIT-502 LOW")
      { S7_Templates := "time_type := Time" } "IEC_Timer_0_DB_74".TON(pt := T#3S, et =>)
      Move(in := 2, out1 => "INTERLOCK DB"."EDI PARAMETER BUFF"."RIT-502 HIGH/ LOW BUFF")
   END_RUNG
   RUNG wire#w2
      { S7_Templates := "SrcType := Real" } LE_Contact(in1 := "AI SCALING DB".PV."RESISTIVITY CUM TRANSMITTER 502", in2 := "INTERLOCK DB"."EDI SET PARAMETER"."RIT-502 HIGH")
      { S7_Templates := "time_type := Time" } "IEC_Timer_0_DB_205".TON(pt := T#2S, et =>)
      Move(in := 1, out1 => "INTERLOCK DB"."EDI PARAMETER BUFF"."RIT-502 HIGH/ LOW BUFF")
   END_RUNG
   RUNG wire#w1
      { S7_Templates := "SrcType := Real" } GT_Contact(in1 := "AI SCALING DB".PV."RESISTIVITY CUM TRANSMITTER 502", in2 := "INTERLOCK DB"."EDI SET PARAMETER"."RIT-502 LOW")
      { S7_Templates := "SrcType := Real" } GT_Contact(in1 := "AI SCALING DB".PV."RESISTIVITY CUM TRANSMITTER 502", in2 := "INTERLOCK DB"."EDI SET PARAMETER"."RIT-502 HIGH")
      wire#w3
      { S7_Templates := "time_type := Time" } "IEC_Timer_0_DB_163".TON(pt := T#3S, et =>)
      Move(in := 0, out1 => "INTERLOCK DB"."EDI PARAMETER BUFF"."RIT-502 HIGH/ LOW BUFF")
   END_RUNG
   RUNG wire#w1
      I_Contact( "EDI DB"."EDI 501B" )
   END_RUNG wire#w3
   RUNG wire#powerrail
      "TIMING_SECS_DB_35"(RESET := wire#w4, INPUT := wire#w5, "SET TIME" := "INTERLOCK DB"."EDI SET TIMER"."RIT-502 HIGH TIMER SET", "PRESENT VALUE OF TIME" => "INTERLOCK DB"."EDI PV TIMER"."RIT-502 HIGH TIMER PV", DONE =>)
   END_RUNG
   RUNG wire#powerrail
      { S7_Templates := "SrcType := Int" } NE_Contact(in1 := "MODE SELECTION DB".EDI."PROCESS BUFF", in2 := 2)
   END_RUNG wire#w4
   RUNG wire#powerrail
      { S7_Templates := "SrcType := Int" } NE_Contact(in1 := "INTERLOCK DB"."EDI PARAMETER BUFF"."RIT-502 HIGH/ LOW BUFF", in2 := 2)
   END_RUNG wire#w4
   RUNG wire#powerrail
      { S7_Templates := "SrcType := Int" } EQ_Contact(in1 := "MODE SELECTION DB".EDI."MODE BUFF", in2 := 1)
      { S7_Templates := "SrcType := Int" } EQ_Contact(in1 := "MODE SELECTION DB".EDI."PROCESS BUFF", in2 := 2)
      { S7_Templates := "SrcType := Int" } EQ_Contact(in1 := "INTERLOCK DB"."EDI PARAMETER BUFF"."RIT-502 HIGH/ LOW BUFF", in2 := 2)
   END_RUNG wire#w5
   // the same network as SCL:
   #_w1 := "MODE SELECTION DB".EDI."MODE BUFF" = 1;
   "IEC_Timer_0_DB_75".TON(IN := #_w1 AND ("MODE SELECTION DB".EDI."PROCESS BUFF" = 2) AND "EDI DB"."EDI 501B",
                           PT := T#3S);
   "IEC_Timer_0_DB_74".TON(IN := "IEC_Timer_0_DB_75".Q AND ("AI SCALING DB".PV."RESISTIVITY CUM TRANSMITTER 502" <= "INTERLOCK DB"."EDI SET PARAMETER"."RIT-502 LOW"),
                           PT := T#3S);
   IF "IEC_Timer_0_DB_74".Q THEN "INTERLOCK DB"."EDI PARAMETER BUFF"."RIT-502 HIGH/ LOW BUFF" := 2; END_IF;
   "IEC_Timer_0_DB_205".TON(IN := "IEC_Timer_0_DB_75".Q AND ("AI SCALING DB".PV."RESISTIVITY CUM TRANSMITTER 502" <= "INTERLOCK DB"."EDI SET PARAMETER"."RIT-502 HIGH"),
                           PT := T#2S);
   IF "IEC_Timer_0_DB_205".Q THEN "INTERLOCK DB"."EDI PARAMETER BUFF"."RIT-502 HIGH/ LOW BUFF" := 1; END_IF;
   "IEC_Timer_0_DB_163".TON(IN := #_w1 AND ((("AI SCALING DB".PV."RESISTIVITY CUM TRANSMITTER 502" > "INTERLOCK DB"."EDI SET PARAMETER"."RIT-502 LOW") AND ("AI SCALING DB".PV."RESISTIVITY CUM TRANSMITTER 502" > "INTERLOCK DB"."EDI SET PARAMETER"."RIT-502 HIGH")) OR NOT "EDI DB"."EDI 501B"),
                           PT := T#3S);
   IF "IEC_Timer_0_DB_163".Q THEN "INTERLOCK DB"."EDI PARAMETER BUFF"."RIT-502 HIGH/ LOW BUFF" := 0; END_IF;
   "TIMING_SECS_DB_35"("SET TIME" := "INTERLOCK DB"."EDI SET TIMER"."RIT-502 HIGH TIMER SET",   // "TIMING_SECS"
                       RESET := ("MODE SELECTION DB".EDI."PROCESS BUFF" <> 2) OR ("INTERLOCK DB"."EDI PARAMETER BUFF"."RIT-502 HIGH/ LOW BUFF" <> 2),
                       INPUT := ("MODE SELECTION DB".EDI."MODE BUFF" = 1) AND ("MODE SELECTION DB".EDI."PROCESS BUFF" = 2) AND ("INTERLOCK DB"."EDI PARAMETER BUFF"."RIT-502 HIGH/ LOW BUFF" = 2),
                       "PRESENT VALUE OF TIME" => "INTERLOCK DB"."EDI PV TIMER"."RIT-502 HIGH TIMER PV");
END_REGION
END_FUNCTION
